C05501=1157.629,21.828,-48.363,-179.973,6.133,149.097
C05502=1157.624,22.077,-48.378,-179.970,6.134,149.096
C05503=1157.618,22.327,-48.393,-179.968,6.134,149.095
C05504=1157.613,22.576,-48.407,-179.966,6.135,149.095
C05505=1157.608,22.826,-48.421,-179.962,6.136,149.094
C05506=1157.603,23.076,-48.435,-179.960,6.137,149.094
C05507=1157.598,23.326,-48.450,-179.958,6.138,149.093
C05508=1157.593,23.575,-48.465,-179.955,6.138,149.093
C05509=1157.588,23.824,-48.479,-179.952,6.140,149.092
C05510=1157.583,24.074,-48.493,-179.950,6.140,149.092
C05511=1157.578,24.323,-48.507,-179.947,6.141,149.091
C05512=1157.573,24.573,-48.521,-179.945,6.142,149.090
C05513=1157.567,24.822,-48.537,-179.942,6.143,149.090
C05514=1157.562,25.072,-48.551,-179.940,6.144,149.089
C05515=1157.557,25.322,-48.566,-179.937,6.144,149.089
C05516=1157.552,25.571,-48.580,-179.935,6.145,149.088
C05517=1157.548,25.820,-48.595,-179.932,6.146,149.087
C05518=1157.543,26.070,-48.609,-179.930,6.147,149.087
C05519=1157.537,26.319,-48.624,-179.927,6.148,149.086
C05520=1157.532,26.569,-48.638,-179.924,6.149,149.086
C05521=1157.527,26.818,-48.653,-179.922,6.150,149.085
C05522=1157.522,27.068,-48.667,-179.919,6.151,149.085
C05523=1157.517,27.318,-48.681,-179.917,6.151,149.084
C05524=1157.511,27.587,-48.698,-179.914,6.153,149.084
C05525=1157.506,27.856,-48.713,-179.911,6.153,149.083
C05526=1157.501,28.124,-48.729,-179.908,6.155,149.082
C05527=1157.495,28.393,-48.745,-179.906,6.155,149.082
C05528=1157.490,28.643,-48.760,-179.903,6.156,149.081
C05529=1157.485,28.893,-48.774,-179.900,6.158,149.081
C05530=1157.481,29.142,-48.789,-179.898,6.158,149.080
C05531=1157.475,29.392,-48.804,-179.896,6.159,149.080
C05532=1157.470,29.640,-48.819,-179.892,6.160,149.079
C05533=1157.465,29.890,-48.833,-179.890,6.161,149.078
C05534=1157.460,30.140,-48.847,-179.888,6.161,149.078
C05535=1157.454,30.389,-48.863,-179.885,6.162,149.077
C05536=1157.449,30.639,-48.877,-179.882,6.164,149.077
C05537=1157.445,30.888,-48.892,-179.880,6.164,149.076
C05538=1157.439,31.138,-48.907,-179.877,6.165,149.076
C05539=1157.434,31.387,-48.922,-179.875,6.166,149.075
C05540=1157.429,31.637,-48.936,-179.872,6.167,149.074
C05541=1157.424,31.887,-48.950,-179.870,6.168,149.074
C05542=1157.419,32.136,-48.966,-179.867,6.169,149.073
C05543=1157.414,32.386,-48.980,-179.864,6.170,149.073
C05544=1157.409,32.635,-48.995,-179.862,6.170,149.072
C05545=1157.404,32.885,-49.010,-179.860,6.171,149.072
C05546=1157.399,33.134,-49.025,-179.856,6.172,149.071
C05547=1157.394,33.383,-49.040,-179.854,6.173,149.071
C05548=1157.389,33.633,-49.055,-179.852,6.174,149.070
C05549=1157.384,33.882,-49.070,-179.849,6.175,149.069
C05550=1157.378,34.132,-49.085,-179.846,6.176,149.069
C05551=1157.374,34.381,-49.100,-179.844,6.177,149.068
C05552=1157.369,34.631,-49.114,-179.841,6.178,149.068
C05553=1157.364,34.881,-49.130,-179.839,6.179,149.067
C05554=1157.359,35.131,-49.144,-179.836,6.179,149.066
C05555=1157.354,35.380,-49.160,-179.833,6.181,149.066
C05556=1157.349,35.629,-49.175,-179.831,6.182,149.066
C05557=1157.344,35.879,-49.189,-179.828,6.182,149.065
C05558=1157.339,36.128,-49.205,-179.826,6.184,149.064
C05559=1157.334,36.377,-49.220,-179.823,6.184,149.064
C05560=1157.328,36.627,-49.235,-179.821,6.185,149.063
C05561=1157.324,36.876,-49.250,-179.818,6.187,149.063
C05562=1157.318,37.126,-49.265,-179.815,6.187,149.062
C05563=1157.313,37.376,-49.279,-179.813,6.188,149.062
C05564=1157.308,37.625,-49.295,-179.810,6.190,149.061
C05565=1157.303,37.874,-49.310,-179.807,6.190,149.060
C05566=1157.298,38.124,-49.325,-179.805,6.191,149.060
C05567=1157.294,38.374,-49.340,-179.802,6.192,149.059
C05568=1157.288,38.623,-49.356,-179.800,6.193,149.059
C05569=1157.283,38.873,-49.370,-179.797,6.193,149.058
C05570=1157.278,39.122,-49.386,-179.794,6.195,149.058
C05571=1157.273,39.372,-49.401,-179.792,6.196,149.057
C05572=1157.268,39.621,-49.416,-179.790,6.196,149.057
C05573=1157.263,39.871,-49.431,-179.786,6.198,149.056
C05574=1157.257,40.120,-49.446,-179.784,6.199,149.055
C05575=1157.253,40.369,-49.461,-179.782,6.199,149.055
C05576=1157.248,40.619,-49.477,-179.779,6.201,149.054
C05577=1157.243,40.868,-49.492,-179.777,6.202,149.054
C05578=1157.238,41.118,-49.507,-179.774,6.202,149.053
C05579=1157.233,41.367,-49.522,-179.771,6.204,149.053
C05580=1157.228,41.617,-49.538,-179.769,6.204,149.052
C05581=1157.222,41.866,-49.553,-179.766,6.206,149.052
C05582=1157.218,42.116,-49.569,-179.763,6.206,149.051
C05583=1157.213,42.365,-49.584,-179.761,6.207,149.051
C05584=1157.208,42.615,-49.599,-179.758,6.208,149.050
C05585=1157.203,42.865,-49.614,-179.756,6.209,149.049
C05586=1157.197,43.114,-49.630,-179.753,6.210,149.049
C05587=1157.192,43.363,-49.645,-179.750,6.211,149.048
C05588=1157.188,43.613,-49.661,-179.748,6.212,149.048
C05589=1157.183,43.862,-49.676,-179.745,6.214,149.047
C05590=1157.178,44.112,-49.691,-179.743,6.214,149.047
C05591=1157.172,44.361,-49.707,-179.740,6.215,149.046
C05592=1157.168,44.610,-49.722,-179.737,6.217,149.046
C05593=1157.163,44.860,-49.738,-179.735,6.217,149.045
C05594=1157.157,45.110,-49.753,-179.733,6.218,149.045
C05595=1157.153,45.359,-49.768,-179.729,6.219,149.044
C05596=1157.147,45.608,-49.784,-179.727,6.220,149.043
C05597=1157.143,45.858,-49.800,-179.724,6.221,149.043
C05598=1157.138,46.107,-49.815,-179.722,6.222,149.042
C05599=1157.133,46.357,-49.830,-179.719,6.223,149.042
C05600=1157.127,46.606,-49.846,-179.716,6.224,149.041
C05601=1157.123,46.856,-49.861,-179.714,6.225,149.041
C05602=1157.118,47.105,-49.877,-179.711,6.226,149.040
C05603=1157.112,47.355,-49.892,-179.709,6.227,149.040
C05604=1157.107,47.604,-49.908,-179.706,6.228,149.039
C05605=1157.103,47.854,-49.923,-179.704,6.229,149.039
C05606=1157.098,48.103,-49.939,-179.701,6.230,149.038
C05607=1157.092,48.353,-49.955,-179.698,6.232,149.037
C05608=1157.088,48.602,-49.970,-179.695,6.232,149.037
C05609=1157.083,48.852,-49.986,-179.693,6.233,149.036
C05610=1157.077,49.101,-50.001,-179.690,6.234,149.036
C05611=1157.072,49.350,-50.017,-179.688,6.235,149.035
C05612=1157.068,49.600,-50.033,-179.685,6.237,149.035
C05613=1157.063,49.849,-50.048,-179.683,6.237,149.034
C05614=1157.057,50.099,-50.064,-179.680,6.239,149.034
C05615=1157.053,50.349,-50.080,-179.677,6.239,149.033
C05616=1157.047,50.598,-50.096,-179.675,6.240,149.033
C05617=1157.043,50.847,-50.110,-179.672,6.241,149.032
C05618=1157.038,51.096,-50.127,-179.670,6.242,149.031
C05619=1157.033,51.346,-50.143,-179.666,6.244,149.031
C05620=1157.027,51.596,-50.158,-179.664,6.244,149.030
C05621=1157.022,51.845,-50.174,-179.661,6.246,149.030
C05622=1157.018,52.094,-50.191,-179.659,6.247,149.029
C05623=1157.013,52.344,-50.206,-179.657,6.247,149.029
C05624=1157.008,52.594,-50.222,-179.653,6.249,149.028
C05625=1157.003,52.843,-50.237,-179.651,6.250,149.028
C05626=1156.998,53.092,-50.253,-179.648,6.251,149.027
C05627=1156.993,53.342,-50.269,-179.646,6.252,149.027
C05628=1156.987,53.610,-50.286,-179.643,6.253,149.026
C05629=1156.982,53.879,-50.303,-179.641,6.254,149.025
C05630=1156.976,54.147,-50.320,-179.637,6.255,149.025
C05631=1156.971,54.416,-50.337,-179.634,6.256,149.024
C05632=1156.966,54.666,-50.353,-179.632,6.257,149.024
C05633=1156.961,54.915,-50.370,-179.629,6.259,149.023
C05634=1156.957,55.165,-50.385,-179.627,6.259,149.023
C05635=1156.951,55.414,-50.401,-179.624,6.260,149.022
C05636=1156.946,55.663,-50.417,-179.621,6.262,149.021
C05637=1156.941,55.913,-50.433,-179.619,6.263,149.021
C05638=1156.936,56.162,-50.449,-179.616,6.264,149.021
C05639=1156.932,56.412,-50.465,-179.614,6.265,149.020
C05640=1156.926,56.661,-50.481,-179.611,6.266,149.019
C05641=1156.921,56.910,-50.497,-179.608,6.267,149.019
C05642=1156.916,57.160,-50.513,-179.605,6.268,149.018
C05643=1156.911,57.409,-50.529,-179.603,6.269,149.018
C05644=1156.906,57.659,-50.545,-179.600,6.271,149.017
C05645=1156.901,57.908,-50.561,-179.598,6.271,149.017
C05646=1156.897,58.158,-50.578,-179.595,6.273,149.016
C05647=1156.891,58.407,-50.593,-179.593,6.274,149.016
C05648=1156.887,58.657,-50.610,-179.589,6.275,149.015
C05649=1156.881,58.906,-50.625,-179.587,6.276,149.015
C05650=1156.876,59.155,-50.642,-179.584,6.277,149.014
C05651=1156.871,59.405,-50.658,-179.582,6.278,149.014
C05652=1156.866,59.654,-50.674,-179.580,6.279,149.013
C05653=1156.862,59.904,-50.690,-179.576,6.280,149.012
C05654=1156.856,60.153,-50.706,-179.574,6.281,149.012
C05655=1156.852,60.403,-50.722,-179.571,6.282,149.011
C05656=1156.847,60.652,-50.738,-179.569,6.283,149.011
C05657=1156.841,60.902,-50.755,-179.566,6.285,149.010
C05658=1156.836,61.151,-50.771,-179.564,6.285,149.010
C05659=1156.832,61.400,-50.788,-179.561,6.287,149.009
C05660=1156.826,61.650,-50.804,-179.558,6.287,149.009
C05661=1156.822,61.899,-50.820,-179.555,6.289,149.008
C05662=1156.816,62.148,-50.836,-179.553,6.290,149.008
C05663=1156.812,62.398,-50.852,-179.550,6.291,149.007
C05664=1156.807,62.647,-50.869,-179.548,6.292,149.007
C05665=1156.802,62.897,-50.885,-179.545,6.293,149.006
C05666=1156.796,63.146,-50.902,-179.542,6.294,149.006
C05667=1156.792,63.395,-50.918,-179.539,6.296,149.005
C05668=1156.787,63.646,-50.934,-179.537,6.296,149.005
C05669=1156.782,63.894,-50.951,-179.534,6.298,149.004
C05670=1156.777,64.144,-50.967,-179.532,6.299,149.003
C05671=1156.772,64.393,-50.983,-179.529,6.300,149.003
C05672=1156.767,64.643,-50.999,-179.526,6.301,149.002
C05673=1156.762,64.892,-51.016,-179.524,6.302,149.002
C05674=1156.757,65.142,-51.032,-179.521,6.304,149.001
C05675=1156.752,65.391,-51.049,-179.518,6.305,149.001
C05676=1156.747,65.640,-51.065,-179.516,6.306,149.000
C05677=1156.743,65.890,-51.082,-179.513,6.307,149.000
C05678=1156.737,66.139,-51.098,-179.510,6.308,148.999
C05679=1156.732,66.389,-51.115,-179.508,6.309,148.999
C05680=1156.727,66.638,-51.131,-179.505,6.311,148.998
C05681=1156.723,66.887,-51.148,-179.503,6.312,148.998
C05682=1156.717,67.137,-51.165,-179.500,6.313,148.997
C05683=1156.712,67.386,-51.181,-179.497,6.314,148.997
C05684=1156.708,67.636,-51.197,-179.494,6.315,148.996
C05685=1156.703,67.885,-51.214,-179.492,6.316,148.996
C05686=1156.697,68.134,-51.231,-179.489,6.318,148.995
C05687=1156.693,68.384,-51.248,-179.487,6.318,148.995
C05688=1156.688,68.633,-51.264,-179.484,6.320,148.994
C05689=1156.683,68.882,-51.281,-179.481,6.321,148.994
C05690=1156.678,69.133,-51.297,-179.478,6.322,148.993
C05691=1156.673,69.381,-51.313,-179.476,6.324,148.993
C05692=1156.668,69.631,-51.330,-179.473,6.324,148.992
C05693=1156.663,69.881,-51.347,-179.470,6.326,148.991
C05694=1156.658,70.129,-51.364,-179.468,6.327,148.991
C05695=1156.653,70.379,-51.380,-179.465,6.328,148.991
C05696=1156.648,70.629,-51.398,-179.463,6.329,148.990
C05697=1156.643,70.877,-51.414,-179.460,6.330,148.989
C05698=1156.639,71.127,-51.431,-179.457,6.332,148.989
C05699=1156.633,71.377,-51.448,-179.455,6.333,148.988
C05700=1156.628,71.625,-51.464,-179.452,6.334,148.988
C05701=1156.624,71.875,-51.481,-179.449,6.335,148.987
C05702=1156.619,72.125,-51.498,-179.447,6.336,148.987
C05703=1156.613,72.374,-51.514,-179.444,6.337,148.986
C05704=1156.608,72.623,-51.532,-179.441,6.339,148.986
C05705=1156.604,72.873,-51.548,-179.438,6.340,148.985
C05706=1156.599,73.122,-51.565,-179.436,6.341,148.985
C05707=1156.593,73.371,-51.582,-179.433,6.342,148.984
C05708=1156.589,73.621,-51.599,-179.431,6.343,148.984
C05709=1156.584,73.871,-51.616,-179.428,6.345,148.983
C05710=1156.579,74.119,-51.632,-179.426,6.346,148.983
C05711=1156.573,74.369,-51.649,-179.423,6.347,148.982
C05712=1156.569,74.619,-51.666,-179.420,6.349,148.982
C05713=1156.565,74.868,-51.683,-179.417,6.349,148.981
C05714=1156.559,75.117,-51.700,-179.415,6.351,148.981
C05715=1156.555,75.366,-51.717,-179.412,6.352,148.980
C05716=1156.549,75.616,-51.734,-179.409,6.353,148.980
C05717=1156.545,75.865,-51.751,-179.407,6.355,148.979
C05718=1156.539,76.115,-51.768,-179.404,6.355,148.979
C05719=1156.535,76.364,-51.784,-179.401,6.357,148.978
C05720=1156.530,76.613,-51.802,-179.399,6.358,148.978
C05721=1156.525,76.863,-51.819,-179.396,6.359,148.977
C05722=1156.520,77.113,-51.836,-179.393,6.361,148.977
C05723=1156.515,77.361,-51.853,-179.390,6.361,148.976
C05724=1156.510,77.611,-51.870,-179.388,6.363,148.976
C05725=1156.505,77.860,-51.887,-179.386,6.364,148.975
C05726=1156.500,78.110,-51.905,-179.382,6.365,148.975
C05727=1156.495,78.360,-51.922,-179.380,6.367,148.974
C05728=1156.490,78.608,-51.938,-179.378,6.368,148.974
C05729=1156.485,78.857,-51.956,-179.374,6.369,148.973
C05730=1156.481,79.107,-51.973,-179.372,6.370,148.973
C05731=1156.475,79.357,-51.990,-179.369,6.372,148.972
C05732=1156.470,79.625,-52.008,-179.366,6.373,148.971
C05733=1156.465,79.893,-52.027,-179.363,6.375,148.971
C05734=1156.460,80.162,-52.046,-179.361,6.375,148.970
C05735=1156.454,80.430,-52.064,-179.358,6.377,148.970
C05736=1156.449,80.679,-52.081,-179.355,6.378,148.969
C05737=1156.444,80.929,-52.099,-179.352,6.380,148.969
C05738=1156.440,81.178,-52.116,-179.350,6.381,148.968
C05739=1156.435,81.428,-52.133,-179.347,6.382,148.968
C05740=1156.430,81.677,-52.151,-179.345,6.383,148.967
C05741=1156.425,81.927,-52.167,-179.342,6.385,148.967
C05742=1156.420,82.175,-52.185,-179.339,6.386,148.966
C05743=1156.414,82.425,-52.202,-179.337,6.387,148.966
C05744=1156.410,82.674,-52.219,-179.334,6.389,148.965
C05745=1156.405,82.923,-52.237,-179.331,6.390,148.965
C05746=1156.400,83.173,-52.254,-179.328,6.391,148.964
C05747=1156.396,83.422,-52.272,-179.326,6.392,148.964
C05748=1156.390,83.672,-52.289,-179.322,6.394,148.963
C05749=1156.385,83.921,-52.307,-179.320,6.395,148.963
C05750=1156.381,84.171,-52.324,-179.318,6.396,148.962
C05751=1156.376,84.420,-52.342,-179.314,6.398,148.962
C05752=1156.370,84.669,-52.358,-179.312,6.399,148.961
C05753=1156.365,84.918,-52.376,-179.310,6.400,148.961
C05754=1156.361,85.168,-52.393,-179.306,6.402,148.960
C05755=1156.356,85.417,-52.411,-179.304,6.402,148.960
C05756=1156.351,85.666,-52.428,-179.301,6.404,148.959
C05757=1156.346,85.916,-52.446,-179.298,6.405,148.959
C05758=1156.341,86.165,-52.463,-179.296,6.406,148.958
C05759=1156.336,86.414,-52.481,-179.293,6.408,148.958
C05760=1156.332,86.663,-52.499,-179.291,6.410,148.958
C05761=1156.326,86.913,-52.516,-179.288,6.410,148.957
C05762=1156.321,87.162,-52.534,-179.285,6.412,148.956
C05763=1156.317,87.412,-52.551,-179.283,6.414,148.956
C05764=1156.312,87.661,-52.569,-179.280,6.414,148.955
C05765=1156.307,87.910,-52.587,-179.277,6.416,148.955
C05766=1156.302,88.160,-52.604,-179.274,6.417,148.955
C05767=1156.297,88.409,-52.622,-179.272,6.418,148.954
C05768=1156.293,88.658,-52.639,-179.269,6.420,148.954
C05769=1156.288,88.908,-52.657,-179.266,6.421,148.953
C05770=1156.283,89.157,-52.675,-179.264,6.422,148.952
C05771=1156.278,89.406,-52.693,-179.261,6.424,148.952
C05772=1156.273,89.656,-52.710,-179.258,6.425,148.952
C05773=1156.268,89.905,-52.728,-179.256,6.426,148.951
C05774=1156.263,90.154,-52.746,-179.253,6.427,148.951
C05775=1156.258,90.404,-52.764,-179.250,6.429,148.950
C05776=1156.253,90.653,-52.781,-179.248,6.430,148.950
C05777=1156.248,90.902,-52.799,-179.245,6.431,148.949
C05778=1156.243,91.151,-52.817,-179.242,6.433,148.949
C05779=1156.239,91.401,-52.834,-179.239,6.435,148.948
C05780=1156.233,91.650,-52.852,-179.237,6.436,148.948
C05781=1156.228,91.900,-52.870,-179.234,6.437,148.947
C05782=1156.224,92.149,-52.888,-179.231,6.439,148.947
C05783=1156.219,92.398,-52.906,-179.229,6.439,148.946
C05784=1156.214,92.647,-52.924,-179.226,6.441,148.946
C05785=1156.209,92.897,-52.941,-179.223,6.442,148.945
C05786=1156.204,93.147,-52.959,-179.220,6.444,148.945
C05787=1156.199,93.396,-52.977,-179.218,6.445,148.944
C05788=1156.194,93.645,-52.995,-179.215,6.446,148.944
C05789=1156.189,93.894,-53.013,-179.212,6.448,148.943
C05790=1156.185,94.143,-53.031,-179.210,6.449,148.943
C05791=1156.180,94.393,-53.049,-179.207,6.450,148.942
C05792=1156.175,94.642,-53.067,-179.204,6.452,148.942
C05793=1156.170,94.891,-53.085,-179.202,6.454,148.941
C05794=1156.165,95.141,-53.102,-179.199,6.455,148.941
C05795=1156.160,95.390,-53.120,-179.196,6.456,148.940
C05796=1156.155,95.640,-53.139,-179.193,6.458,148.940
C05797=1156.150,95.889,-53.157,-179.191,6.459,148.940
C05798=1156.146,96.138,-53.175,-179.189,6.460,148.939
C05799=1156.141,96.387,-53.193,-179.185,6.461,148.938
C05800=1156.136,96.637,-53.211,-179.183,6.463,148.938
C05801=1156.131,96.886,-53.229,-179.180,6.465,148.938
C05802=1156.126,97.135,-53.247,-179.178,6.466,148.937
C05803=1156.122,97.385,-53.265,-179.175,6.467,148.937
C05804=1156.117,97.634,-53.283,-179.172,6.469,148.936
C05805=1156.112,97.883,-53.301,-179.170,6.470,148.936
C05806=1156.106,98.133,-53.319,-179.167,6.471,148.935
C05807=1156.102,98.381,-53.338,-179.164,6.473,148.935
C05808=1156.097,98.630,-53.356,-179.161,6.474,148.934
C05809=1156.092,98.880,-53.375,-179.158,6.476,148.934
C05810=1156.087,99.129,-53.392,-179.156,6.477,148.933
C05811=1156.082,99.379,-53.410,-179.153,6.478,148.933
C05812=1156.078,99.628,-53.428,-179.150,6.480,148.932
C05813=1156.072,99.877,-53.447,-179.148,6.482,148.932
C05814=1156.068,100.127,-53.465,-179.145,6.483,148.932
C05815=1156.063,100.376,-53.483,-179.142,6.484,148.931
C05816=1156.058,100.625,-53.502,-179.139,6.486,148.931
C05817=1156.053,100.874,-53.520,-179.137,6.487,148.930
C05818=1156.048,101.123,-53.538,-179.135,6.488,148.930
C05819=1156.043,101.373,-53.557,-179.131,6.490,148.929
C05820=1156.038,101.623,-53.575,-179.129,6.491,148.929
C05821=1156.034,101.871,-53.594,-179.126,6.493,148.928
C05822=1156.029,102.120,-53.612,-179.123,6.495,148.928
C05823=1156.024,102.371,-53.631,-179.121,6.495,148.927
C05824=1156.019,102.620,-53.649,-179.118,6.497,148.927
C05825=1156.014,102.868,-53.667,-179.115,6.499,148.926
C05826=1156.009,103.117,-53.685,-179.112,6.500,148.926
C05827=1156.004,103.368,-53.704,-179.110,6.501,148.925
C05828=1155.999,103.617,-53.722,-179.107,6.502,148.925
C05829=1155.995,103.865,-53.741,-179.104,6.504,148.924
C05830=1155.990,104.114,-53.759,-179.102,6.506,148.924
C05831=1155.985,104.365,-53.778,-179.099,6.508,148.924
C05832=1155.980,104.613,-53.796,-179.096,6.508,148.923
C05833=1155.975,104.862,-53.814,-179.094,6.510,148.923
C05834=1155.970,105.113,-53.833,-179.091,6.511,148.922
C05835=1155.966,105.361,-53.852,-179.088,6.513,148.922
C05836=1155.960,105.629,-53.871,-179.085,6.514,148.921
C05837=1155.955,105.898,-53.891,-179.082,6.516,148.921
C05838=1155.951,106.166,-53.912,-179.079,6.518,148.920
C05839=1155.945,106.435,-53.932,-179.076,6.519,148.920
C05840=1155.940,106.684,-53.950,-179.074,6.521,148.919
C05841=1155.935,106.934,-53.970,-179.071,6.523,148.919
C05842=1155.930,107.183,-53.988,-179.068,6.523,148.918
C05843=1155.926,107.431,-54.006,-179.065,6.525,148.918
C05844=1155.920,107.682,-54.025,-179.063,6.527,148.917
C05845=1155.916,107.930,-54.044,-179.060,6.528,148.917
C05846=1155.911,108.179,-54.062,-179.057,6.530,148.917
C05847=1155.906,108.429,-54.081,-179.055,6.530,148.916
C05848=1155.901,108.678,-54.100,-179.052,6.532,148.916
C05849=1155.896,108.928,-54.118,-179.049,6.534,148.915
C05850=1155.892,109.177,-54.137,-179.047,6.536,148.915
C05851=1155.886,109.426,-54.156,-179.044,6.537,148.914
C05852=1155.882,109.676,-54.175,-179.041,6.539,148.914
C05853=1155.877,109.924,-54.193,-179.038,6.540,148.913
C05854=1155.872,110.174,-54.212,-179.036,6.541,148.913
C05855=1155.868,110.423,-54.231,-179.033,6.543,148.912
C05856=1155.862,110.672,-54.250,-179.030,6.545,148.912
C05857=1155.858,110.922,-54.269,-179.028,6.546,148.912
C05858=1155.853,111.170,-54.288,-179.024,6.548,148.911
C05859=1155.848,111.420,-54.306,-179.022,6.549,148.911
C05860=1155.843,111.669,-54.326,-179.020,6.550,148.910
C05861=1155.838,111.918,-54.344,-179.017,6.552,148.910
C05862=1155.833,112.168,-54.363,-179.014,6.554,148.909
C05863=1155.829,112.416,-54.382,-179.011,6.555,148.909
C05864=1155.824,112.667,-54.401,-179.008,6.557,148.908
C05865=1155.819,112.915,-54.420,-179.005,6.558,148.908
C05866=1155.814,113.164,-54.439,-179.003,6.559,148.908
C05867=1155.809,113.414,-54.458,-179.001,6.561,148.907
C05868=1155.804,113.663,-54.477,-178.998,6.563,148.907
C05869=1155.799,113.912,-54.496,-178.995,6.564,148.906
C05870=1155.795,114.161,-54.515,-178.992,6.566,148.906
C05871=1155.790,114.411,-54.534,-178.989,6.567,148.905
C05872=1155.785,114.660,-54.553,-178.987,6.569,148.905
C05873=1155.780,114.909,-54.572,-178.984,6.571,148.904
C05874=1155.775,115.158,-54.592,-178.982,6.572,148.904
C05875=1155.771,115.408,-54.610,-178.978,6.573,148.903
C05876=1155.765,115.657,-54.629,-178.976,6.575,148.903
C05877=1155.761,115.906,-54.649,-178.973,6.577,148.903
C05878=1155.756,116.155,-54.667,-178.970,6.578,148.902
C05879=1155.751,116.405,-54.687,-178.968,6.580,148.902
C05880=1155.747,116.653,-54.706,-178.965,6.582,148.901
C05881=1155.742,116.903,-54.725,-178.962,6.583,148.901
C05882=1155.736,117.152,-54.744,-178.960,6.584,148.900
C05883=1155.732,117.401,-54.763,-178.957,6.586,148.900
C05884=1155.727,117.650,-54.782,-178.954,6.587,148.900
C05885=1155.722,117.900,-54.802,-178.951,6.589,148.899
C05886=1155.718,118.148,-54.821,-178.949,6.591,148.899
C05887=1155.713,118.398,-54.840,-178.946,6.592,148.898
C05888=1155.708,118.648,-54.860,-178.943,6.594,148.898
C05889=1155.703,118.896,-54.879,-178.940,6.596,148.897
C05890=1155.699,119.146,-54.898,-178.937,6.597,148.897
C05891=1155.693,119.395,-54.918,-178.935,6.599,148.897
C05892=1155.689,119.644,-54.937,-178.932,6.600,148.896
C05893=1155.683,119.893,-54.957,-178.930,6.602,148.896
C05894=1155.679,120.142,-54.976,-178.927,6.603,148.895
C05895=1155.675,120.392,-54.995,-178.924,6.605,148.895
C05896=1155.669,120.641,-55.015,-178.921,6.606,148.894
C05897=1155.665,120.890,-55.034,-178.918,6.608,148.894
C05898=1155.660,121.139,-55.053,-178.916,6.610,148.893
C05899=1155.655,121.388,-55.073,-178.913,6.611,148.893
C05900=1155.650,121.638,-55.092,-178.910,6.613,148.893
C05901=1155.645,121.887,-55.112,-178.908,6.615,148.892
C05902=1155.640,122.136,-55.131,-178.905,6.617,148.892
C05903=1155.636,122.385,-55.150,-178.902,6.618,148.891
C05904=1155.631,122.634,-55.170,-178.899,6.619,148.891
C05905=1155.626,122.884,-55.189,-178.897,6.621,148.890
C05906=1155.621,123.133,-55.209,-178.894,6.622,148.890
C05907=1155.616,123.383,-55.228,-178.891,6.624,148.890
C05908=1155.612,123.631,-55.249,-178.889,6.626,148.889
C05909=1155.607,123.880,-55.267,-178.886,6.627,148.889
C05910=1155.602,124.130,-55.287,-178.883,6.629,148.888
C05911=1155.598,124.379,-55.307,-178.880,6.631,148.888
C05912=1155.592,124.628,-55.326,-178.877,6.632,148.887
C05913=1155.588,124.878,-55.346,-178.875,6.634,148.887
C05914=1155.583,125.127,-55.366,-178.872,6.636,148.887
C05915=1155.578,125.375,-55.385,-178.869,6.637,148.886
C05916=1155.573,125.625,-55.405,-178.866,6.639,148.886
C05917=1155.569,125.874,-55.424,-178.864,6.641,148.885
C05918=1155.564,126.122,-55.444,-178.861,6.642,148.885
C05919=1155.559,126.372,-55.464,-178.858,6.644,148.885
C05920=1155.554,126.622,-55.483,-178.856,6.646,148.884
C05921=1155.550,126.871,-55.503,-178.853,6.648,148.884
C05922=1155.545,127.119,-55.523,-178.850,6.648,148.883
C05923=1155.540,127.369,-55.543,-178.848,6.650,148.883
C05924=1155.535,127.619,-55.562,-178.845,6.652,148.882
C05925=1155.531,127.868,-55.583,-178.842,6.653,148.882
C05926=1155.525,128.116,-55.602,-178.839,6.655,148.882
C05927=1155.521,128.366,-55.622,-178.837,6.657,148.881
C05928=1155.516,128.615,-55.642,-178.834,6.658,148.881
C05929=1155.512,128.864,-55.662,-178.831,6.660,148.880
C05930=1155.506,129.113,-55.682,-178.829,6.662,148.880
C05931=1155.502,129.362,-55.701,-178.826,6.664,148.880
C05932=1155.497,129.612,-55.721,-178.823,6.665,148.879
C05933=1155.493,129.861,-55.741,-178.820,6.667,148.879
C05934=1155.487,130.110,-55.761,-178.817,6.668,148.878
C05935=1155.483,130.359,-55.781,-178.814,6.670,148.878
C05936=1155.478,130.608,-55.801,-178.812,6.672,148.877
C05937=1155.474,130.857,-55.821,-178.809,6.673,148.877
C05938=1155.468,131.107,-55.841,-178.806,6.675,148.877
C05939=1155.463,131.356,-55.861,-178.804,6.677,148.876
C05940=1155.458,131.624,-55.882,-178.801,6.679,148.876
C05941=1155.453,131.893,-55.903,-178.798,6.681,148.876
C05942=1155.448,132.162,-55.925,-178.794,6.682,148.875
C05943=1155.443,132.430,-55.947,-178.792,6.684,148.874
C05944=1155.437,132.679,-55.967,-178.789,6.686,148.874
C05945=1155.433,132.928,-55.988,-178.786,6.688,148.874
C05946=1155.428,133.178,-56.007,-178.784,6.689,148.873
C05947=1155.424,133.427,-56.028,-178.781,6.691,148.873
C05948=1155.419,133.675,-56.048,-178.778,6.693,148.873
C05949=1155.414,133.925,-56.067,-178.775,6.695,148.872
C05950=1155.410,134.174,-56.088,-178.773,6.696,148.872
C05951=1155.404,134.424,-56.108,-178.770,6.698,148.871
C05952=1155.400,134.672,-56.128,-178.767,6.700,148.871
C05953=1155.395,134.921,-56.149,-178.765,6.701,148.871
C05954=1155.391,135.171,-56.168,-178.762,6.703,148.870
C05955=1155.386,135.419,-56.188,-178.759,6.705,148.870
C05956=1155.380,135.668,-56.209,-178.756,6.707,148.869
C05957=1155.376,135.918,-56.229,-178.754,6.708,148.869
C05958=1155.371,136.167,-56.249,-178.751,6.710,148.869
C05959=1155.367,136.416,-56.270,-178.748,6.712,148.868
C05960=1155.362,136.665,-56.291,-178.746,6.713,148.868
C05961=1155.357,136.915,-56.310,-178.742,6.715,148.867
C05962=1155.352,137.164,-56.331,-178.740,6.717,148.867
C05963=1155.348,137.413,-56.351,-178.737,6.718,148.866
C05964=1155.343,137.662,-56.372,-178.734,6.720,148.866
C05965=1155.338,137.912,-56.392,-178.731,6.722,148.866
C05966=1155.333,138.160,-56.412,-178.728,6.724,148.865
C05967=1155.329,138.409,-56.432,-178.726,6.726,148.865
C05968=1155.323,138.658,-56.453,-178.723,6.728,148.865
C05969=1155.319,138.907,-56.473,-178.720,6.729,148.864
C05970=1155.314,139.156,-56.493,-178.717,6.731,148.864
C05971=1155.309,139.406,-56.514,-178.715,6.733,148.863
C05972=1155.305,139.655,-56.534,-178.712,6.735,148.863
C05973=1155.300,139.904,-56.555,-178.709,6.736,148.863
C05974=1155.295,140.153,-56.576,-178.707,6.738,148.862
C05975=1155.291,140.402,-56.596,-178.704,6.740,148.862
C05976=1155.286,140.651,-56.616,-178.701,6.741,148.861
C05977=1155.281,140.900,-56.637,-178.699,6.743,148.861
C05978=1155.276,141.150,-56.657,-178.696,6.745,148.861
C05979=1155.271,141.399,-56.678,-178.693,6.747,148.860
C05980=1155.267,141.648,-56.698,-178.690,6.748,148.860
C05981=1155.262,141.897,-56.719,-178.688,6.750,148.859
C05982=1155.257,142.146,-56.740,-178.684,6.753,148.859
C05983=1155.253,142.395,-56.760,-178.682,6.754,148.859
C05984=1155.247,142.644,-56.781,-178.679,6.756,148.858
C05985=1155.243,142.893,-56.801,-178.676,6.758,148.858
C05986=1155.238,143.142,-56.822,-178.674,6.759,148.858
C05987=1155.233,143.391,-56.843,-178.671,6.761,148.857
C05988=1155.229,143.640,-56.863,-178.668,6.763,148.857
C05989=1155.224,143.890,-56.884,-178.665,6.765,148.856
C05990=1155.219,144.139,-56.904,-178.663,6.766,148.856
C05991=1155.214,144.387,-56.926,-178.660,6.768,148.856
C05992=1155.211,144.637,-56.947,-178.657,6.770,148.855
C05993=1155.205,144.886,-56.968,-178.655,6.772,148.855
C05994=1155.201,145.135,-56.988,-178.652,6.774,148.855
C05995=1155.196,145.384,-57.009,-178.649,6.776,148.854
C05996=1155.191,145.633,-57.030,-178.646,6.778,148.854
C05997=1155.186,145.883,-57.051,-178.644,6.780,148.854
C05998=1155.182,146.131,-57.071,-178.641,6.781,148.853
C05999=1155.177,146.381,-57.092,-178.638,6.783,148.853
C06000=1155.172,146.629,-57.113,-178.636,6.785,148.852
C06001=1155.167,146.878,-57.134,-178.633,6.787,148.852
C06002=1155.162,147.128,-57.155,-178.630,6.788,148.852
C06003=1155.158,147.377,-57.176,-178.627,6.790,148.851
C06004=1155.153,147.627,-57.197,-178.624,6.792,148.851
C06005=1155.149,147.875,-57.218,-178.621,6.794,148.850
C06006=1155.144,148.124,-57.239,-178.619,6.796,148.850
C06007=1155.139,148.373,-57.260,-178.616,6.798,148.850
C06008=1155.134,148.622,-57.280,-178.613,6.799,148.849
C06009=1155.129,148.871,-57.302,-178.611,6.801,148.849
C06010=1155.125,149.120,-57.322,-178.608,6.803,148.849
C06011=1155.120,149.370,-57.343,-178.605,6.805,148.848
C06012=1155.115,149.618,-57.365,-178.602,6.807,148.848
C06013=1155.111,149.867,-57.385,-178.599,6.809,148.847
C06014=1155.106,150.117,-57.406,-178.597,6.811,148.847
C06015=1155.101,150.365,-57.428,-178.594,6.813,148.847
C06016=1155.096,150.614,-57.448,-178.592,6.814,148.847
C06017=1155.092,150.864,-57.470,-178.589,6.816,148.846
C06018=1155.087,151.113,-57.491,-178.586,6.818,148.846
C06019=1155.083,151.362,-57.512,-178.583,6.820,148.845
C06020=1155.077,151.611,-57.533,-178.580,6.822,148.845
C06021=1155.073,151.860,-57.554,-178.577,6.824,148.845
C06022=1155.068,152.110,-57.576,-178.575,6.826,148.844
C06023=1155.064,152.358,-57.597,-178.572,6.827,148.844
C06024=1155.059,152.607,-57.618,-178.569,6.829,148.843
C06025=1155.054,152.856,-57.640,-178.567,6.831,148.843
C06026=1155.049,153.105,-57.661,-178.563,6.833,148.843
C06027=1155.045,153.354,-57.682,-178.561,6.835,148.842
C06028=1155.040,153.603,-57.703,-178.558,6.837,148.842
C06029=1155.035,153.852,-57.725,-178.556,6.839,148.842
C06030=1155.030,154.101,-57.746,-178.553,6.841,148.841
C06031=1155.026,154.350,-57.767,-178.550,6.842,148.841
C06032=1155.021,154.600,-57.788,-178.547,6.845,148.841
C06033=1155.016,154.848,-57.810,-178.544,6.847,148.840
C06034=1155.011,155.098,-57.831,-178.542,6.848,148.840
C06035=1155.007,155.347,-57.853,-178.539,6.850,148.840
C06036=1155.002,155.596,-57.874,-178.536,6.852,148.839
C06037=1154.998,155.844,-57.895,-178.534,6.854,148.839
C06038=1154.993,156.094,-57.917,-178.531,6.856,148.839
C06039=1154.988,156.343,-57.938,-178.528,6.858,148.838
C06040=1154.983,156.592,-57.959,-178.525,6.860,148.838
C06041=1154.978,156.841,-57.980,-178.523,6.862,148.838
C06042=1154.974,157.090,-58.002,-178.520,6.863,148.837
C06043=1154.969,157.339,-58.024,-178.517,6.866,148.837
C06044=1154.964,157.608,-58.047,-178.514,6.868,148.836
C06045=1154.959,157.877,-58.070,-178.511,6.869,148.836
C06046=1154.954,158.146,-58.094,-178.508,6.872,148.836
C06047=1154.949,158.415,-58.117,-178.505,6.874,148.835
C06048=1154.945,158.664,-58.138,-178.503,6.875,148.835
C06049=1154.939,158.913,-58.159,-178.499,6.878,148.835
C06050=1154.935,159.162,-58.181,-178.497,6.880,148.834
C06051=1154.930,159.411,-58.203,-178.494,6.882,148.834
C06052=1154.926,159.660,-58.225,-178.492,6.883,148.834
C06053=1154.921,159.909,-58.246,-178.488,6.886,148.833
C06054=1154.916,160.158,-58.268,-178.486,6.888,148.833
C06055=1154.912,160.407,-58.290,-178.483,6.889,148.833
C06056=1154.907,160.656,-58.311,-178.480,6.891,148.832
C06057=1154.902,160.905,-58.333,-178.478,6.893,148.832
C06058=1154.898,161.154,-58.355,-178.474,6.896,148.831
C06059=1154.893,161.403,-58.376,-178.472,6.898,148.831
C06060=1154.888,161.653,-58.398,-178.469,6.899,148.831
C06061=1154.883,161.901,-58.420,-178.467,6.901,148.831
C06062=1154.879,162.150,-58.441,-178.464,6.903,148.830
C06063=1154.874,162.399,-58.463,-178.461,6.905,148.830
C06064=1154.869,162.648,-58.485,-178.458,6.907,148.829
C06065=1154.865,162.897,-58.507,-178.456,6.909,148.829
C06066=1154.860,163.146,-58.529,-178.453,6.911,148.829
C06067=1154.856,163.395,-58.551,-178.450,6.913,148.829
C06068=1154.850,163.644,-58.573,-178.447,6.915,148.828
C06069=1154.846,163.893,-58.595,-178.444,6.917,148.828
C06070=1154.841,164.142,-58.617,-178.442,6.919,148.827
C06071=1154.836,164.391,-58.639,-178.439,6.922,148.827
C06072=1154.832,164.640,-58.661,-178.436,6.923,148.827
C06073=1154.827,164.889,-58.682,-178.434,6.925,148.827
C06074=1154.823,165.138,-58.704,-178.431,6.927,148.826
C06075=1154.818,165.387,-58.726,-178.428,6.929,148.826
C06076=1154.814,165.636,-58.748,-178.425,6.931,148.825
C06077=1154.808,165.885,-58.770,-178.423,6.933,148.825
C06078=1154.804,166.134,-58.792,-178.420,6.935,148.825
C06079=1154.799,166.383,-58.814,-178.417,6.937,148.825
C06080=1154.795,166.632,-58.836,-178.414,6.939,148.824
C06081=1154.790,166.881,-58.858,-178.411,6.941,148.824
C06082=1154.786,167.130,-58.880,-178.409,6.943,148.824
C06083=1154.780,167.379,-58.902,-178.406,6.946,148.823
C06084=1154.776,167.628,-58.925,-178.403,6.947,148.823
C06085=1154.771,167.877,-58.947,-178.400,6.949,148.823
C06086=1154.767,168.126,-58.969,-178.398,6.951,148.822
C06087=1154.761,168.375,-58.991,-178.395,6.954,148.822
C06088=1154.757,168.624,-59.013,-178.392,6.955,148.822
C06089=1154.752,168.873,-59.035,-178.389,6.957,148.821
C06090=1154.748,169.122,-59.057,-178.387,6.959,148.821
C06091=1154.743,169.371,-59.080,-178.383,6.961,148.821
C06092=1154.738,169.620,-59.102,-178.381,6.964,148.820
C06093=1154.734,169.869,-59.124,-178.379,6.965,148.820
C06094=1154.730,170.117,-59.146,-178.375,6.968,148.820
C06095=1154.725,170.367,-59.169,-178.373,6.970,148.819
C06096=1154.720,170.616,-59.191,-178.370,6.971,148.819
C06097=1154.715,170.865,-59.213,-178.368,6.973,148.819
C06098=1154.710,171.113,-59.236,-178.364,6.976,148.819
C06099=1154.706,171.363,-59.258,-178.362,6.978,148.818
C06100=1154.702,171.612,-59.280,-178.359,6.979,148.818
C06101=1154.696,171.860,-59.303,-178.356,6.982,148.818
C06102=1154.692,172.110,-59.325,-178.354,6.984,148.817
C06103=1154.687,172.358,-59.347,-178.351,6.986,148.817
C06104=1154.682,172.607,-59.370,-178.348,6.988,148.817
C06105=1154.678,172.857,-59.392,-178.345,6.991,148.816
C06106=1154.674,173.105,-59.414,-178.343,6.992,148.816
C06107=1154.669,173.354,-59.437,-178.340,6.994,148.816
C06108=1154.665,173.603,-59.460,-178.337,6.997,148.815
C06109=1154.659,173.852,-59.482,-178.334,6.999,148.815
C06110=1154.655,174.101,-59.504,-178.332,7.000,148.815
C06111=1154.650,174.350,-59.527,-178.328,7.003,148.814
C06112=1154.645,174.599,-59.549,-178.326,7.005,148.814
C06113=1154.641,174.848,-59.572,-178.324,7.007,148.814
C06114=1154.636,175.097,-59.594,-178.320,7.009,148.814
C06115=1154.632,175.345,-59.617,-178.318,7.011,148.813
C06116=1154.627,175.595,-59.639,-178.315,7.013,148.813
C06117=1154.623,175.844,-59.662,-178.312,7.016,148.813
C06118=1154.617,176.093,-59.684,-178.309,7.017,148.812
C06119=1154.613,176.341,-59.707,-178.307,7.019,148.812
C06120=1154.608,176.590,-59.731,-178.303,7.022,148.812
C06121=1154.604,176.839,-59.752,-178.301,7.024,148.812
C06122=1154.599,177.088,-59.776,-178.299,7.026,148.811
C06123=1154.595,177.337,-59.798,-178.295,7.028,148.811
C06124=1154.590,177.586,-59.821,-178.293,7.030,148.811
C06125=1154.585,177.834,-59.843,-178.290,7.032,148.810
C06126=1154.580,178.084,-59.866,-178.287,7.035,148.810
C06127=1154.576,178.333,-59.889,-178.284,7.036,148.810
C06128=1154.571,178.581,-59.912,-178.282,7.038,148.809
C06129=1154.567,178.831,-59.934,-178.279,7.041,148.809
C06130=1154.562,179.080,-59.957,-178.276,7.043,148.809
C06131=1154.557,179.329,-59.981,-178.274,7.045,148.809
C06132=1154.553,179.578,-60.003,-178.271,7.047,148.808
C06133=1154.548,179.826,-60.026,-178.268,7.049,148.808
C06134=1154.544,180.075,-60.048,-178.265,7.051,148.808
C06135=1154.539,180.324,-60.072,-178.263,7.054,148.807
C06136=1154.534,180.574,-60.094,-178.260,7.056,148.807
C06137=1154.530,180.822,-60.117,-178.257,7.058,148.807
C06138=1154.525,181.071,-60.140,-178.254,7.060,148.807
C06139=1154.521,181.319,-60.163,-178.252,7.062,148.806
C06140=1154.516,181.568,-60.186,-178.248,7.064,148.806
C06141=1154.511,181.818,-60.209,-178.246,7.067,148.806
C06142=1154.507,182.066,-60.231,-178.243,7.068,148.805
C06143=1154.502,182.315,-60.255,-178.240,7.071,148.805
C06144=1154.497,182.564,-60.278,-178.238,7.073,148.805
C06145=1154.493,182.813,-60.301,-178.235,7.076,148.805
C06146=1154.489,183.062,-60.324,-178.232,7.077,148.804
C06147=1154.484,183.311,-60.348,-178.229,7.079,148.804
C06148=1154.479,183.581,-60.373,-178.227,7.082,148.804
C06149=1154.474,183.850,-60.397,-178.223,7.085,148.803
C06150=1154.469,184.120,-60.422,-178.221,7.086,148.803
C06151=1154.463,184.390,-60.447,-178.217,7.089,148.803
C06152=1154.459,184.638,-60.470,-178.215,7.091,148.803
C06153=1154.455,184.887,-60.493,-178.212,7.094,148.802
C06154=1154.450,185.137,-60.517,-178.209,7.095,148.802
C06155=1154.445,185.385,-60.540,-178.206,7.098,148.802
C06156=1154.441,185.634,-60.562,-178.204,7.100,148.801
C06157=1154.436,185.883,-60.586,-178.201,7.102,148.801
C06158=1154.431,186.132,-60.609,-178.198,7.105,148.801
C06159=1154.427,186.381,-60.632,-178.195,7.106,148.801
C06160=1154.422,186.630,-60.656,-178.192,7.109,148.800
C06161=1154.417,186.879,-60.679,-178.190,7.111,148.800
C06162=1154.414,187.127,-60.703,-178.187,7.113,148.800
C06163=1154.409,187.376,-60.726,-178.184,7.115,148.799
C06164=1154.404,187.625,-60.749,-178.182,7.117,148.799
C06165=1154.400,187.874,-60.773,-178.179,7.120,148.799
C06166=1154.394,188.122,-60.796,-178.176,7.122,148.799
C06167=1154.390,188.371,-60.819,-178.173,7.125,148.798
C06168=1154.385,188.620,-60.842,-178.170,7.126,148.798
C06169=1154.381,188.869,-60.865,-178.168,7.128,148.798
C06170=1154.376,189.117,-60.889,-178.165,7.131,148.798
C06171=1154.372,189.366,-60.913,-178.162,7.133,148.797
C06172=1154.367,189.616,-60.936,-178.159,7.136,148.797
C06173=1154.362,189.865,-60.959,-178.157,7.137,148.797
C06174=1154.358,190.114,-60.983,-178.154,7.140,148.797
C06175=1154.353,190.362,-61.007,-178.151,7.142,148.796
C06176=1154.349,190.611,-61.030,-178.149,7.144,148.796
C06177=1154.344,190.860,-61.053,-178.146,7.147,148.796
C06178=1154.339,191.109,-61.077,-178.143,7.149,148.795
C06179=1154.335,191.358,-61.101,-178.140,7.151,148.795
C06180=1154.330,191.607,-61.124,-178.138,7.153,148.795
C06181=1154.325,191.856,-61.148,-178.134,7.156,148.795
C06182=1154.321,192.104,-61.172,-178.132,7.158,148.795
C06183=1154.316,192.353,-61.195,-178.129,7.160,148.794
C06184=1154.312,192.602,-61.218,-178.127,7.163,148.794
C06185=1154.307,192.850,-61.242,-178.124,7.164,148.794
C06186=1154.302,193.099,-61.266,-178.121,7.167,148.793
C06187=1154.298,193.349,-61.289,-178.118,7.169,148.793
C06188=1154.293,193.597,-61.313,-178.115,7.172,148.793
C06189=1154.289,193.846,-61.337,-178.113,7.174,148.793
C06190=1154.284,194.094,-61.361,-178.110,7.176,148.792
C06191=1154.280,194.343,-61.384,-178.107,7.178,148.792
C06192=1154.275,194.592,-61.408,-178.104,7.181,148.792
C06193=1154.271,194.842,-61.432,-178.102,7.183,148.792
C06194=1154.266,195.091,-61.455,-178.099,7.186,148.792
C06195=1154.261,195.339,-61.480,-178.096,7.187,148.791
C06196=1154.257,195.588,-61.503,-178.093,7.190,148.791
C06197=1154.252,195.837,-61.527,-178.091,7.192,148.791
C06198=1154.247,196.086,-61.551,-178.088,7.195,148.791
C06199=1154.243,196.334,-61.575,-178.085,7.197,148.790
C06200=1154.239,196.583,-61.599,-178.082,7.198,148.790
C06201=1154.234,196.832,-61.622,-178.080,7.201,148.790
C06202=1154.230,197.080,-61.646,-178.077,7.203,148.789
C06203=1154.225,197.330,-61.671,-178.074,7.206,148.789
C06204=1154.220,197.579,-61.695,-178.071,7.208,148.789
C06205=1154.216,197.828,-61.718,-178.069,7.211,148.789
C06206=1154.211,198.076,-61.742,-178.066,7.212,148.789
C06207=1154.207,198.324,-61.766,-178.063,7.215,148.788
C06208=1154.201,198.574,-61.790,-178.061,7.217,148.788
C06209=1154.197,198.822,-61.814,-178.057,7.220,148.788
C06210=1154.193,199.071,-61.839,-178.055,7.222,148.788
C06211=1154.189,199.320,-61.862,-178.052,7.224,148.787
C06212=1154.184,199.569,-61.886,-178.050,7.226,148.787
C06213=1154.179,199.817,-61.911,-178.046,7.229,148.787
C06214=1154.174,200.066,-61.934,-178.044,7.231,148.787
C06215=1154.171,200.316,-61.959,-178.041,7.234,148.786
C06216=1154.166,200.564,-61.983,-178.039,7.236,148.786
C06217=1154.161,200.813,-62.007,-178.035,7.238,148.786
C06218=1154.156,201.062,-62.031,-178.033,7.241,148.786
C06219=1154.152,201.310,-62.055,-178.030,7.243,148.785
C06220=1154.147,201.560,-62.080,-178.027,7.246,148.785
C06221=1154.143,201.808,-62.104,-178.024,7.248,148.785
C06222=1154.139,202.056,-62.128,-178.022,7.251,148.785
C06223=1154.133,202.306,-62.152,-178.019,7.252,148.785
C06224=1154.129,202.554,-62.176,-178.016,7.255,148.784
C06225=1154.125,202.803,-62.200,-178.013,7.257,148.784
C06226=1154.120,203.052,-62.225,-178.011,7.260,148.784
C06227=1154.115,203.300,-62.249,-178.008,7.262,148.784
C06228=1154.112,203.550,-62.274,-178.005,7.265,148.784
C06229=1154.107,203.798,-62.298,-178.003,7.266,148.783
C06230=1154.102,204.047,-62.322,-178.000,7.269,148.783
C06231=1154.098,204.295,-62.346,-177.997,7.271,148.783
C06232=1154.093,204.544,-62.371,-177.994,7.274,148.783
C06233=1154.088,204.794,-62.395,-177.991,7.277,148.782
C06234=1154.083,205.042,-62.419,-177.989,7.279,148.782
C06235=1154.079,205.291,-62.444,-177.986,7.281,148.782
C06236=1154.074,205.540,-62.469,-177.983,7.283,148.782
C06237=1154.070,205.788,-62.493,-177.980,7.286,148.781
C06238=1154.065,206.037,-62.517,-177.978,7.288,148.781
C06239=1154.061,206.286,-62.542,-177.975,7.291,148.781
C06240=1154.057,206.535,-62.566,-177.972,7.293,148.781
C06241=1154.052,206.783,-62.591,-177.970,7.296,148.781
C06242=1154.048,207.032,-62.616,-177.966,7.298,148.780
C06243=1154.043,207.281,-62.640,-177.964,7.300,148.780
C06244=1154.039,207.529,-62.664,-177.961,7.303,148.780
C06245=1154.034,207.779,-62.689,-177.959,7.305,148.780
C06246=1154.029,208.027,-62.714,-177.955,7.308,148.780
C06247=1154.025,208.276,-62.738,-177.953,7.310,148.779
C06248=1154.020,208.525,-62.763,-177.950,7.312,148.779
C06249=1154.016,208.773,-62.787,-177.947,7.315,148.779
C06250=1154.011,209.022,-62.813,-177.944,7.317,148.779
C06251=1154.007,209.271,-62.837,-177.942,7.320,148.779
C06252=1154.002,209.541,-62.864,-177.938,7.323,148.778
C06253=1153.997,209.812,-62.891,-177.936,7.325,148.778
C06254=1153.992,210.082,-62.918,-177.933,7.327,148.778
C06255=1153.987,210.353,-62.945,-177.930,7.330,148.778
C06256=1153.982,210.602,-62.969,-177.927,7.333,148.777
C06257=1153.977,210.850,-62.994,-177.925,7.335,148.777
C06258=1153.974,211.099,-63.018,-177.922,7.338,148.777
C06259=1153.969,211.347,-63.044,-177.919,7.340,148.777
C06260=1153.964,211.597,-63.069,-177.916,7.342,148.777
C06261=1153.960,211.845,-63.093,-177.913,7.345,148.776
C06262=1153.955,212.093,-63.118,-177.911,7.347,148.776
C06263=1153.950,212.343,-63.143,-177.908,7.350,148.776
C06264=1153.946,212.591,-63.167,-177.905,7.353,148.776
C06265=1153.942,212.840,-63.193,-177.903,7.355,148.776
C06266=1153.937,213.089,-63.218,-177.899,7.357,148.775
C06267=1153.933,213.338,-63.242,-177.897,7.359,148.775
C06268=1153.928,213.586,-63.268,-177.894,7.362,148.775
C06269=1153.924,213.835,-63.293,-177.891,7.365,148.775
C06270=1153.919,214.083,-63.318,-177.889,7.367,148.775
C06271=1153.915,214.333,-63.343,-177.886,7.370,148.774
C06272=1153.910,214.581,-63.367,-177.883,7.373,148.774
C06273=1153.906,214.830,-63.393,-177.881,7.375,148.774
C06274=1153.901,215.079,-63.417,-177.878,7.377,148.774
C06275=1153.897,215.327,-63.443,-177.875,7.379,148.774
C06276=1153.892,215.576,-63.467,-177.872,7.382,148.774
C06277=1153.888,215.825,-63.493,-177.869,7.385,148.773
C06278=1153.882,216.074,-63.518,-177.867,7.387,148.773
C06279=1153.879,216.322,-63.543,-177.864,7.390,148.773
C06280=1153.874,216.571,-63.568,-177.861,7.392,148.773
C06281=1153.870,216.820,-63.593,-177.859,7.395,148.773
C06282=1153.865,217.068,-63.619,-177.856,7.397,148.772
C06283=1153.860,217.317,-63.644,-177.853,7.400,148.772
C06284=1153.856,217.565,-63.669,-177.850,7.402,148.772
C06285=1153.852,217.814,-63.694,-177.847,7.405,148.772
C06286=1153.847,218.062,-63.719,-177.845,7.407,148.772
C06287=1153.843,218.311,-63.745,-177.842,7.409,148.772
C06288=1153.838,218.561,-63.770,-177.839,7.412,148.771
C06289=1153.833,218.809,-63.795,-177.837,7.414,148.771
C06290=1153.829,219.058,-63.821,-177.834,7.417,148.771
C06291=1153.824,219.306,-63.846,-177.831,7.420,148.771
C06292=1153.820,219.555,-63.871,-177.829,7.422,148.771
C06293=1153.816,219.804,-63.897,-177.825,7.425,148.770
C06294=1153.811,220.052,-63.921,-177.823,7.428,148.770
C06295=1153.807,220.301,-63.947,-177.820,7.430,148.770
C06296=1153.802,220.549,-63.972,-177.817,7.432,148.770
C06297=1153.798,220.798,-63.998,-177.814,7.435,148.770
C06298=1153.793,221.047,-64.024,-177.812,7.437,148.770
C06299=1153.788,221.296,-64.049,-177.809,7.440,148.769
C06300=1153.784,221.544,-64.074,-177.806,7.443,148.769
C06301=1153.780,221.793,-64.100,-177.804,7.445,148.769
C06302=1153.775,222.041,-64.125,-177.801,7.448,148.769
C06303=1153.771,222.290,-64.151,-177.798,7.450,148.769
C06304=1153.766,222.539,-64.176,-177.795,7.453,148.769
C06305=1153.762,222.788,-64.202,-177.792,7.455,148.768
C06306=1153.757,223.036,-64.227,-177.790,7.458,148.768
C06307=1153.752,223.285,-64.253,-177.787,7.461,148.768
C06308=1153.748,223.533,-64.279,-177.784,7.463,148.768
C06309=1153.744,223.782,-64.304,-177.781,7.466,148.768
C06310=1153.740,224.031,-64.330,-177.779,7.469,148.768
C06311=1153.735,224.279,-64.355,-177.776,7.471,148.768
C06312=1153.731,224.528,-64.381,-177.773,7.473,148.767
C06313=1153.727,224.777,-64.407,-177.770,7.476,148.767
C06314=1153.722,225.025,-64.432,-177.768,7.478,148.767
C06315=1153.717,225.274,-64.459,-177.765,7.481,148.767
C06316=1153.712,225.523,-64.484,-177.762,7.484,148.767
C06317=1153.708,225.771,-64.510,-177.759,7.487,148.767
C06318=1153.703,226.020,-64.536,-177.757,7.489,148.766
C06319=1153.699,226.268,-64.561,-177.754,7.492,148.766
C06320=1153.695,226.517,-64.587,-177.751,7.494,148.766
C06321=1153.690,226.765,-64.612,-177.749,7.497,148.766
C06322=1153.685,227.014,-64.639,-177.746,7.499,148.766
C06323=1153.681,227.263,-64.664,-177.743,7.502,148.766
C06324=1153.677,227.512,-64.690,-177.740,7.505,148.766
C06325=1153.672,227.760,-64.716,-177.738,7.507,148.765
C06326=1153.668,228.009,-64.741,-177.735,7.510,148.765
C06327=1153.664,228.257,-64.768,-177.732,7.513,148.765
C06328=1153.659,228.506,-64.794,-177.729,7.516,148.765
C06329=1153.655,228.755,-64.820,-177.727,7.518,148.765
C06330=1153.650,229.003,-64.845,-177.724,7.520,148.765
C06331=1153.646,229.252,-64.871,-177.721,7.523,148.764
C06332=1153.641,229.500,-64.898,-177.718,7.526,148.764
C06333=1153.637,229.749,-64.924,-177.716,7.528,148.764
C06334=1153.632,229.998,-64.950,-177.713,7.531,148.764
C06335=1153.628,230.246,-64.975,-177.710,7.534,148.764
C06336=1153.623,230.495,-65.002,-177.707,7.537,148.764
C06337=1153.619,230.744,-65.028,-177.705,7.539,148.764
C06338=1153.615,230.992,-65.054,-177.702,7.541,148.763
C06339=1153.610,231.241,-65.080,-177.699,7.544,148.763
C06340=1153.605,231.489,-65.106,-177.696,7.547,148.763
C06341=1153.601,231.738,-65.132,-177.694,7.549,148.763
C06342=1153.596,231.987,-65.158,-177.691,7.552,148.763
C06343=1153.592,232.235,-65.185,-177.688,7.555,148.763
C06344=1153.588,232.484,-65.210,-177.685,7.558,148.763
C06345=1153.583,232.732,-65.237,-177.683,7.560,148.762
C06346=1153.579,232.981,-65.263,-177.680,7.563,148.762
C06347=1153.575,233.230,-65.289,-177.677,7.565,148.762
C06348=1153.569,233.478,-65.316,-177.674,7.568,148.762
C06349=1153.565,233.727,-65.341,-177.672,7.571,148.762
C06350=1153.561,233.975,-65.368,-177.669,7.573,148.762
C06351=1153.556,234.224,-65.394,-177.666,7.576,148.762
C06352=1153.552,234.472,-65.421,-177.663,7.579,148.761
C06353=1153.547,234.721,-65.447,-177.660,7.582,148.761
C06354=1153.543,234.969,-65.473,-177.658,7.584,148.761
C06355=1153.538,235.218,-65.500,-177.655,7.587,148.761
C06356=1153.534,235.490,-65.529,-177.652,7.590,148.761
C06357=1153.529,235.762,-65.557,-177.649,7.592,148.761
C06358=1153.524,236.033,-65.586,-177.646,7.596,148.761
C06359=1153.519,236.305,-65.615,-177.643,7.599,148.761
C06360=1153.515,236.554,-65.641,-177.640,7.601,148.760
C06361=1153.510,236.802,-65.668,-177.638,7.604,148.760
C06362=1153.506,237.051,-65.694,-177.635,7.607,148.760
C06363=1153.501,237.299,-65.721,-177.632,7.610,148.760
C06364=1153.497,237.548,-65.747,-177.629,7.613,148.760
C06365=1153.492,237.797,-65.774,-177.627,7.615,148.760
C06366=1153.489,238.045,-65.800,-177.624,7.617,148.760
C06367=1153.484,238.293,-65.827,-177.621,7.620,148.760
C06368=1153.479,238.543,-65.854,-177.618,7.623,148.760
C06369=1153.475,238.791,-65.880,-177.615,7.626,148.759
C06370=1153.470,239.039,-65.907,-177.613,7.628,148.759
C06371=1153.466,239.288,-65.933,-177.610,7.631,148.759
C06372=1153.461,239.536,-65.960,-177.607,7.634,148.759
C06373=1153.458,239.785,-65.986,-177.604,7.637,148.759
C06374=1153.453,240.033,-66.013,-177.602,7.640,148.759
C06375=1153.448,240.282,-66.040,-177.599,7.643,148.759
C06376=1153.444,240.530,-66.066,-177.597,7.645,148.759
C06377=1153.439,240.779,-66.093,-177.594,7.648,148.759
C06378=1153.435,241.027,-66.120,-177.591,7.651,148.758
C06379=1153.431,241.276,-66.147,-177.588,7.653,148.758
C06380=1153.426,241.524,-66.174,-177.585,7.656,148.758
C06381=1153.421,241.773,-66.200,-177.582,7.659,148.758
C06382=1153.417,242.021,-66.227,-177.580,7.661,148.758
C06383=1153.413,242.270,-66.254,-177.577,7.664,148.758
C06384=1153.409,242.519,-66.281,-177.575,7.667,148.758
C06385=1153.405,242.767,-66.308,-177.572,7.670,148.758
C06386=1153.400,243.016,-66.335,-177.569,7.673,148.758
C06387=1153.395,243.264,-66.362,-177.566,7.676,148.757
C06388=1153.391,243.512,-66.388,-177.564,7.678,148.757
C06389=1153.387,243.761,-66.415,-177.561,7.681,148.757
C06390=1153.382,244.009,-66.442,-177.558,7.684,148.757
C06391=1153.377,244.258,-66.469,-177.555,7.686,148.757
C06392=1153.374,244.506,-66.496,-177.552,7.689,148.757
C06393=1153.369,244.755,-66.523,-177.550,7.692,148.757
C06394=1153.365,245.004,-66.550,-177.547,7.694,148.757
C06395=1153.360,245.252,-66.577,-177.545,7.697,148.757
C06396=1153.355,245.501,-66.605,-177.541,7.700,148.756
C06397=1153.352,245.749,-66.631,-177.539,7.703,148.756
C06398=1153.347,245.998,-66.658,-177.536,7.706,148.756
C06399=1153.342,246.246,-66.685,-177.533,7.709,148.756
C06400=1153.338,246.495,-66.713,-177.530,7.712,148.756
C06401=1153.334,246.744,-66.740,-177.528,7.714,148.756
C06402=1153.329,246.992,-66.767,-177.525,7.717,148.756
C06403=1153.325,247.240,-66.794,-177.523,7.720,148.756
C06404=1153.321,247.488,-66.821,-177.520,7.723,148.756
C06405=1153.316,247.737,-66.848,-177.517,7.726,148.756
C06406=1153.312,247.986,-66.875,-177.514,7.728,148.756
C06407=1153.307,248.234,-66.902,-177.511,7.731,148.756
C06408=1153.303,248.482,-66.930,-177.509,7.734,148.756
C06409=1153.298,248.731,-66.957,-177.506,7.736,148.755
C06410=1153.294,248.979,-66.984,-177.503,7.739,148.755
C06411=1153.290,249.229,-67.012,-177.500,7.742,148.755
C06412=1153.285,249.476,-67.040,-177.498,7.745,148.755
C06413=1153.281,249.725,-67.066,-177.495,7.748,148.755
C06414=1153.277,249.973,-67.093,-177.492,7.751,148.755
C06415=1153.273,250.222,-67.121,-177.489,7.754,148.755
C06416=1153.268,250.470,-67.148,-177.487,7.757,148.755
C06417=1153.264,250.719,-67.175,-177.484,7.760,148.755
C06418=1153.259,250.967,-67.203,-177.482,7.762,148.755
C06419=1153.255,251.216,-67.231,-177.479,7.765,148.754
C06420=1153.250,251.464,-67.258,-177.476,7.768,148.754
C06421=1153.246,251.712,-67.285,-177.473,7.771,148.754
C06422=1153.241,251.961,-67.312,-177.470,7.774,148.754
C06423=1153.237,252.210,-67.340,-177.468,7.776,148.754
C06424=1153.233,252.458,-67.368,-177.465,7.779,148.754
C06425=1153.228,252.706,-67.395,-177.462,7.782,148.754
C06426=1153.224,252.955,-67.423,-177.459,7.785,148.754
C06427=1153.219,253.204,-67.451,-177.457,7.787,148.754
C06428=1153.215,253.451,-67.478,-177.454,7.790,148.754
C06429=1153.211,253.701,-67.506,-177.452,7.793,148.754
C06430=1153.207,253.948,-67.534,-177.449,7.796,148.754
C06431=1153.202,254.197,-67.561,-177.446,7.799,148.754
C06432=1153.198,254.446,-67.589,-177.443,7.802,148.754
C06433=1153.193,254.694,-67.616,-177.441,7.805,148.754
C06434=1153.189,254.942,-67.644,-177.438,7.808,148.753
C06435=1153.185,255.190,-67.672,-177.435,7.811,148.753
C06436=1153.180,255.439,-67.699,-177.432,7.814,148.753
C06437=1153.176,255.687,-67.727,-177.429,7.817,148.753
C06438=1153.172,255.936,-67.755,-177.427,7.820,148.753
C06439=1153.167,256.184,-67.782,-177.424,7.822,148.753
C06440=1153.163,256.432,-67.810,-177.422,7.825,148.753
C06441=1153.159,256.681,-67.838,-177.419,7.828,148.753
C06442=1153.154,256.930,-67.866,-177.416,7.831,148.753
C06443=1153.150,257.178,-67.894,-177.413,7.834,148.753
C06444=1153.145,257.427,-67.921,-177.411,7.837,148.753
C06445=1153.141,257.674,-67.949,-177.408,7.839,148.753
C06446=1153.137,257.923,-67.977,-177.405,7.842,148.753
C06447=1153.132,258.172,-68.005,-177.402,7.845,148.753
C06448=1153.128,258.420,-68.033,-177.399,7.848,148.753
C06449=1153.124,258.668,-68.061,-177.397,7.851,148.752
C06450=1153.119,258.917,-68.089,-177.394,7.854,148.752
C06451=1153.115,259.165,-68.117,-177.391,7.857,148.752
C06452=1153.110,259.414,-68.144,-177.389,7.860,148.752
C06453=1153.106,259.662,-68.172,-177.386,7.863,148.752
C06454=1153.101,259.910,-68.201,-177.383,7.866,148.752
C06455=1153.098,260.159,-68.229,-177.381,7.869,148.752
C06456=1153.093,260.407,-68.257,-177.378,7.871,148.752
C06457=1153.089,260.656,-68.285,-177.376,7.874,148.752
C06458=1153.084,260.904,-68.312,-177.373,7.877,148.752
C06459=1153.080,261.153,-68.341,-177.370,7.880,148.752
C06460=1153.076,261.426,-68.371,-177.367,7.884,148.752
C06461=1153.071,261.699,-68.403,-177.364,7.887,148.752
C06462=1153.066,261.972,-68.434,-177.361,7.890,148.752
C06463=1153.061,262.246,-68.465,-177.358,7.894,148.752
C06464=1153.056,262.494,-68.493,-177.355,7.896,148.752
C06465=1153.052,262.743,-68.521,-177.352,7.899,148.752
C06466=1153.048,262.990,-68.549,-177.349,7.902,148.752
C06467=1153.044,263.239,-68.578,-177.347,7.905,148.752
C06468=1153.039,263.487,-68.605,-177.344,7.908,148.752
C06469=1153.035,263.736,-68.634,-177.342,7.911,148.752
C06470=1153.030,263.984,-68.662,-177.339,7.914,148.752
C06471=1153.026,264.233,-68.691,-177.336,7.917,148.752
C06472=1153.022,264.481,-68.719,-177.333,7.920,148.752
C06473=1153.017,264.730,-68.747,-177.330,7.923,148.751
C06474=1153.013,264.978,-68.775,-177.328,7.925,148.751
C06475=1153.009,265.226,-68.804,-177.325,7.928,148.751
C06476=1153.005,265.474,-68.833,-177.323,7.931,148.751
C06477=1153.000,265.722,-68.861,-177.320,7.935,148.751
C06478=1152.996,265.971,-68.889,-177.318,7.937,148.751
C06479=1152.991,266.219,-68.917,-177.315,7.940,148.751
C06480=1152.987,266.468,-68.946,-177.312,7.943,148.751
C06481=1152.983,266.716,-68.975,-177.309,7.946,148.751
C06482=1152.979,266.964,-69.003,-177.307,7.949,148.751
C06483=1152.974,267.213,-69.032,-177.304,7.952,148.751
C06484=1152.970,267.461,-69.059,-177.301,7.955,148.751
C06485=1152.965,267.710,-69.088,-177.299,7.958,148.751
C06486=1152.961,267.958,-69.118,-177.296,7.961,148.751
C06487=1152.957,268.206,-69.145,-177.293,7.964,148.751
C06488=1152.952,268.455,-69.174,-177.290,7.967,148.751
C06489=1152.949,268.703,-69.203,-177.288,7.970,148.751
C06490=1152.944,268.951,-69.231,-177.285,7.973,148.751
C06491=1152.939,269.200,-69.260,-177.282,7.976,148.751
C06492=1152.936,269.448,-69.289,-177.280,7.979,148.751
C06493=1152.931,269.696,-69.317,-177.277,7.982,148.751
C06494=1152.926,269.945,-69.346,-177.274,7.985,148.751
C06495=1152.923,270.193,-69.375,-177.271,7.988,148.751
C06496=1152.918,270.441,-69.403,-177.269,7.991,148.751
C06497=1152.913,270.689,-69.433,-177.266,7.994,148.751
C06498=1152.910,270.938,-69.461,-177.264,7.997,148.751
C06499=1152.905,271.186,-69.489,-177.260,8.001,148.751
C06500=1152.900,271.434,-69.519,-177.257,8.004,148.751
C06501=1152.897,271.683,-69.547,-177.255,8.007,148.751
C06502=1152.892,271.930,-69.576,-177.252,8.010,148.751
C06503=1152.887,272.179,-69.605,-177.250,8.013,148.751
C06504=1152.883,272.427,-69.634,-177.247,8.016,148.751
C06505=1152.880,272.676,-69.662,-177.244,8.019,148.751
C06506=1152.875,272.924,-69.691,-177.241,8.022,148.751
C06507=1152.870,273.172,-69.720,-177.239,8.025,148.751
C06508=1152.866,273.421,-69.749,-177.236,8.028,148.751
C06509=1152.863,273.669,-69.778,-177.233,8.031,148.751
C06510=1152.858,273.917,-69.807,-177.231,8.034,148.751
C06511=1152.853,274.165,-69.836,-177.228,8.037,148.751
C06512=1152.849,274.414,-69.865,-177.226,8.040,148.751
C06513=1152.845,274.662,-69.894,-177.223,8.043,148.751
C06514=1152.841,274.910,-69.923,-177.220,8.046,148.751
C06515=1152.836,275.158,-69.952,-177.218,8.049,148.751
C06516=1152.832,275.407,-69.981,-177.215,8.052,148.751
C06517=1152.828,275.655,-70.010,-177.212,8.055,148.751
C06518=1152.823,275.904,-70.039,-177.209,8.058,148.751
C06519=1152.819,276.151,-70.068,-177.207,8.062,148.751
C06520=1152.814,276.400,-70.098,-177.204,8.065,148.751
C06521=1152.811,276.648,-70.127,-177.201,8.067,148.751
C06522=1152.806,276.897,-70.155,-177.199,8.070,148.751
C06523=1152.802,277.145,-70.185,-177.196,8.074,148.751
C06524=1152.798,277.393,-70.214,-177.194,8.077,148.751
C06525=1152.793,277.641,-70.243,-177.190,8.080,148.751
C06526=1152.789,277.889,-70.273,-177.188,8.083,148.751
C06527=1152.785,278.138,-70.302,-177.185,8.087,148.751
C06528=1152.780,278.386,-70.331,-177.182,8.090,148.751
C06529=1152.776,278.634,-70.360,-177.180,8.092,148.751
C06530=1152.772,278.883,-70.390,-177.177,8.096,148.751
C06531=1152.768,279.131,-70.419,-177.175,8.099,148.751
C06532=1152.763,279.378,-70.448,-177.172,8.102,148.751
C06533=1152.759,279.627,-70.478,-177.169,8.105,148.751
C06534=1152.755,279.875,-70.507,-177.167,8.108,148.751
C06535=1152.751,280.123,-70.537,-177.164,8.111,148.751
C06536=1152.746,280.372,-70.566,-177.161,8.114,148.751
C06537=1152.742,280.620,-70.595,-177.159,8.117,148.751
C06538=1152.738,280.869,-70.624,-177.156,8.120,148.751
C06539=1152.734,281.117,-70.654,-177.153,8.124,148.751
C06540=1152.729,281.365,-70.683,-177.150,8.127,148.751
C06541=1152.725,281.613,-70.712,-177.148,8.130,148.751
C06542=1152.720,281.861,-70.742,-177.145,8.133,148.751
C06543=1152.716,282.109,-70.771,-177.143,8.136,148.751
C06544=1152.712,282.357,-70.802,-177.140,8.139,148.751
C06545=1152.708,282.605,-70.831,-177.137,8.142,148.751
C06546=1152.704,282.853,-70.860,-177.134,8.145,148.751
C06547=1152.699,283.102,-70.890,-177.132,8.148,148.751
C06548=1152.695,283.350,-70.920,-177.129,8.151,148.751
C06549=1152.691,283.599,-70.949,-177.127,8.155,148.752
C06550=1152.686,283.847,-70.979,-177.124,8.157,148.751
C06551=1152.682,284.095,-71.008,-177.121,8.161,148.751
C06552=1152.678,284.343,-71.038,-177.118,8.164,148.752
C06553=1152.674,284.591,-71.069,-177.116,8.167,148.752
C06554=1152.669,284.840,-71.098,-177.113,8.170,148.752
C06555=1152.665,285.088,-71.127,-177.111,8.174,148.752
C06556=1152.661,285.336,-71.157,-177.108,8.177,148.752
C06557=1152.657,285.584,-71.187,-177.105,8.180,148.752
C06558=1152.652,285.832,-71.217,-177.103,8.183,148.752
C06559=1152.648,286.081,-71.247,-177.100,8.186,148.752
C06560=1152.644,286.329,-71.276,-177.097,8.190,148.752
C06561=1152.640,286.577,-71.306,-177.094,8.193,148.752
C06562=1152.636,286.825,-71.336,-177.092,8.196,148.752
C06563=1152.631,287.073,-71.366,-177.089,8.199,148.752
C06564=1152.626,287.348,-71.399,-177.086,8.202,148.752
C06565=1152.621,287.624,-71.432,-177.083,8.206,148.752
C06566=1152.617,287.899,-71.465,-177.080,8.210,148.752
C06567=1152.612,288.174,-71.498,-177.077,8.213,148.752
C06568=1152.608,288.422,-71.529,-177.075,8.216,148.752
C06569=1152.603,288.671,-71.558,-177.072,8.219,148.752
C06570=1152.600,288.918,-71.588,-177.069,8.223,148.752
C06571=1152.595,289.167,-71.618,-177.067,8.226,148.753
C06572=1152.591,289.415,-71.648,-177.064,8.229,148.752
C06573=1152.587,289.663,-71.678,-177.062,8.232,148.753
C06574=1152.583,289.911,-71.709,-177.059,8.235,148.753
C06575=1152.578,290.160,-71.739,-177.056,8.238,148.753
C06576=1152.575,290.407,-71.769,-177.054,8.241,148.753
C06577=1152.570,290.656,-71.799,-177.051,8.244,148.753
C06578=1152.566,290.904,-71.829,-177.048,8.248,148.753
C06579=1152.562,291.152,-71.858,-177.045,8.251,148.753
C06580=1152.557,291.400,-71.889,-177.043,8.255,148.753
C06581=1152.553,291.648,-71.919,-177.040,8.258,148.753
C06582=1152.549,291.897,-71.950,-177.037,8.261,148.753
C06583=1152.545,292.145,-71.979,-177.035,8.264,148.753
C06584=1152.540,292.393,-72.010,-177.032,8.267,148.753
C06585=1152.536,292.641,-72.040,-177.029,8.271,148.753
C06586=1152.532,292.889,-72.070,-177.027,8.274,148.753
C06587=1152.527,293.137,-72.100,-177.024,8.277,148.753
C06588=1152.524,293.385,-72.131,-177.022,8.280,148.753
C06589=1152.519,293.634,-72.161,-177.019,8.283,148.754
C06590=1152.515,293.881,-72.191,-177.017,8.286,148.754
C06591=1152.511,294.129,-72.222,-177.014,8.290,148.754
C06592=1152.507,294.377,-72.252,-177.011,8.293,148.754
C06593=1152.502,294.626,-72.282,-177.009,8.297,148.754
C06594=1152.499,294.874,-72.313,-177.006,8.300,148.754
C06595=1152.494,295.122,-72.343,-177.003,8.303,148.754
C06596=1152.489,295.370,-72.374,-177.001,8.306,148.754
C06597=1152.485,295.618,-72.404,-176.998,8.309,148.754
C06598=1152.481,295.867,-72.435,-176.995,8.313,148.754
C06599=1152.477,296.114,-72.465,-176.993,8.316,148.754
C06600=1152.473,296.362,-72.496,-176.990,8.319,148.754
C06601=1152.469,296.610,-72.526,-176.988,8.322,148.754
C06602=1152.465,296.859,-72.557,-176.985,8.325,148.754
C06603=1152.460,297.107,-72.587,-176.982,8.329,148.755
C06604=1152.456,297.355,-72.617,-176.979,8.332,148.755
C06605=1152.451,297.603,-72.648,-176.977,8.336,148.755
C06606=1152.447,297.852,-72.679,-176.974,8.339,148.755
C06607=1152.443,298.099,-72.709,-176.972,8.342,148.755
C06608=1152.439,298.347,-72.740,-176.969,8.345,148.755
C06609=1152.436,298.595,-72.770,-176.966,8.349,148.755
C06610=1152.431,298.843,-72.801,-176.963,8.352,148.755
C06611=1152.426,299.091,-72.832,-176.961,8.355,148.755
C06612=1152.422,299.340,-72.863,-176.959,8.358,148.755
C06613=1152.418,299.588,-72.893,-176.956,8.361,148.755
C06614=1152.414,299.836,-72.924,-176.953,8.365,148.756
C06615=1152.409,300.084,-72.955,-176.950,8.368,148.756
C06616=1152.406,300.332,-72.985,-176.948,8.372,148.756
C06617=1152.401,300.580,-73.016,-176.945,8.375,148.756
C06618=1152.397,300.828,-73.047,-176.943,8.378,148.756
C06619=1152.393,301.077,-73.078,-176.940,8.382,148.756
C06620=1152.389,301.324,-73.109,-176.937,8.385,148.756
C06621=1152.385,301.572,-73.140,-176.935,8.388,148.756
C06622=1152.381,301.820,-73.171,-176.932,8.391,148.756
C06623=1152.376,302.068,-73.202,-176.930,8.394,148.756
C06624=1152.372,302.317,-73.233,-176.927,8.398,148.756
C06625=1152.368,302.564,-73.263,-176.924,8.401,148.757
C06626=1152.364,302.812,-73.294,-176.922,8.405,148.757
C06627=1152.360,303.060,-73.325,-176.919,8.408,148.757
C06628=1152.355,303.308,-73.356,-176.917,8.411,148.757
C06629=1152.350,303.556,-73.387,-176.913,8.415,148.757
C06630=1152.346,303.805,-73.418,-176.911,8.418,148.757
C06631=1152.342,304.052,-73.450,-176.909,8.421,148.757
C06632=1152.339,304.301,-73.480,-176.906,8.424,148.757
C06633=1152.334,304.549,-73.511,-176.903,8.428,148.758
C06634=1152.330,304.796,-73.542,-176.901,8.432,148.758
C06635=1152.326,305.045,-73.574,-176.898,8.435,148.758
C06636=1152.321,305.293,-73.604,-176.896,8.438,148.758
C06637=1152.318,305.541,-73.636,-176.893,8.441,148.758
C06638=1152.313,305.789,-73.667,-176.890,8.445,148.758
C06639=1152.309,306.037,-73.698,-176.888,8.448,148.758
C06640=1152.305,306.285,-73.730,-176.885,8.451,148.758
C06641=1152.301,306.533,-73.761,-176.883,8.454,148.758
C06642=1152.296,306.781,-73.792,-176.880,8.458,148.759
C06643=1152.292,307.029,-73.823,-176.877,8.461,148.759
C06644=1152.288,307.277,-73.854,-176.875,8.465,148.759
C06645=1152.283,307.525,-73.885,-176.872,8.468,148.759
C06646=1152.279,307.773,-73.917,-176.869,8.472,148.759
C06647=1152.275,308.021,-73.948,-176.867,8.475,148.759
C06648=1152.271,308.269,-73.979,-176.864,8.478,148.759
C06649=1152.267,308.517,-74.011,-176.862,8.481,148.759
C06650=1152.263,308.765,-74.042,-176.859,8.484,148.760
C06651=1152.258,309.013,-74.073,-176.856,8.489,148.760
C06652=1152.255,309.261,-74.105,-176.854,8.492,148.760
C06653=1152.250,309.509,-74.136,-176.851,8.495,148.760
C06654=1152.246,309.757,-74.168,-176.849,8.498,148.760
C06655=1152.242,310.005,-74.199,-176.846,8.502,148.760
C06656=1152.238,310.253,-74.230,-176.843,8.505,148.760
C06657=1152.234,310.501,-74.262,-176.841,8.508,148.760
C06658=1152.230,310.749,-74.293,-176.838,8.512,148.761
C06659=1152.225,310.997,-74.325,-176.835,8.515,148.761
C06660=1152.221,311.244,-74.357,-176.833,8.519,148.761
C06661=1152.217,311.493,-74.388,-176.831,8.522,148.761
C06662=1152.213,311.740,-74.420,-176.828,8.526,148.761
C06663=1152.209,311.988,-74.451,-176.825,8.529,148.761
C06664=1152.205,312.237,-74.483,-176.823,8.532,148.761
C06665=1152.201,312.484,-74.514,-176.821,8.536,148.762
C06666=1152.196,312.733,-74.546,-176.817,8.539,148.762
C06667=1152.192,312.980,-74.578,-176.815,8.543,148.762
C06668=1152.188,313.258,-74.614,-176.812,8.547,148.762
C06669=1152.183,313.536,-74.648,-176.809,8.551,148.762
C06670=1152.179,313.813,-74.684,-176.806,8.554,148.762
C06671=1152.174,314.090,-74.719,-176.803,8.558,148.762
C06672=1152.169,314.338,-74.752,-176.801,8.561,148.763
C06673=1152.166,314.586,-74.784,-176.798,8.565,148.763
C06674=1152.161,314.834,-74.815,-176.795,8.568,148.763
C06675=1152.158,315.082,-74.847,-176.793,8.571,148.763
C06676=1152.152,315.330,-74.878,-176.790,8.576,148.763
C06677=1152.149,315.578,-74.910,-176.788,8.579,148.763
C06678=1152.145,315.826,-74.942,-176.785,8.582,148.763
C06679=1152.140,316.074,-74.974,-176.783,8.585,148.764
C06680=1152.136,316.322,-75.006,-176.780,8.589,148.764
C06681=1152.132,316.570,-75.038,-176.778,8.592,148.764
C06682=1152.129,316.818,-75.070,-176.775,8.596,148.764
C06683=1152.124,317.066,-75.102,-176.772,8.599,148.764
C06684=1152.120,317.314,-75.133,-176.770,8.603,148.764
C06685=1152.116,317.562,-75.165,-176.767,8.606,148.765
C06686=1152.111,317.809,-75.197,-176.765,8.609,148.765
C06687=1152.107,318.057,-75.229,-176.762,8.613,148.765
C06688=1152.104,318.305,-75.261,-176.759,8.616,148.765
C06689=1152.100,318.553,-75.294,-176.757,8.620,148.765
C06690=1152.095,318.800,-75.326,-176.754,8.624,148.765
C06691=1152.091,319.049,-75.358,-176.752,8.627,148.766
C06692=1152.087,319.297,-75.390,-176.749,8.630,148.766
C06693=1152.083,319.545,-75.422,-176.747,8.634,148.766
C06694=1152.078,319.792,-75.454,-176.744,8.637,148.766
C06695=1152.075,320.041,-75.486,-176.741,8.641,148.766
C06696=1152.071,320.288,-75.519,-176.739,8.645,148.767
C06697=1152.067,320.536,-75.551,-176.736,8.648,148.767
C06698=1152.062,320.784,-75.583,-176.734,8.651,148.767
C06699=1152.058,321.032,-75.615,-176.731,8.655,148.767
C06700=1152.054,321.280,-75.648,-176.729,8.659,148.767
C06701=1152.050,321.528,-75.680,-176.726,8.662,148.767
C06702=1152.046,321.776,-75.712,-176.723,8.666,148.768
C06703=1152.042,322.023,-75.744,-176.721,8.669,148.768
C06704=1152.037,322.271,-75.777,-176.718,8.672,148.768
C06705=1152.034,322.519,-75.809,-176.716,8.676,148.768
C06706=1152.029,322.768,-75.841,-176.713,8.680,148.768
C06707=1152.026,323.015,-75.874,-176.711,8.683,148.769
C06708=1152.021,323.263,-75.906,-176.708,8.687,148.769
C06709=1152.017,323.511,-75.937,-176.705,8.690,148.769
C06710=1152.013,323.758,-75.971,-176.703,8.693,148.769
C06711=1152.009,324.006,-76.002,-176.700,8.697,148.769
C06712=1152.005,324.254,-76.036,-176.698,8.700,148.769
C06713=1152.001,324.502,-76.067,-176.695,8.704,148.770
C06714=1151.997,324.750,-76.101,-176.692,8.708,148.770
C06715=1151.992,324.998,-76.133,-176.690,8.711,148.770
C06716=1151.989,325.245,-76.165,-176.688,8.714,148.770
C06717=1151.984,325.493,-76.198,-176.685,8.718,148.770
C06718=1151.980,325.741,-76.231,-176.683,8.722,148.771
C06719=1151.977,325.989,-76.263,-176.680,8.725,148.771
C06720=1151.972,326.237,-76.296,-176.677,8.729,148.771
C06721=1151.968,326.485,-76.328,-176.675,8.732,148.771
C06722=1151.965,326.733,-76.361,-176.672,8.735,148.771
C06723=1151.960,326.981,-76.393,-176.669,8.739,148.771
C06724=1151.956,327.229,-76.426,-176.667,8.743,148.772
C06725=1151.952,327.476,-76.458,-176.664,8.747,148.772
C06726=1151.948,327.724,-76.491,-176.662,8.750,148.772
C06727=1151.943,327.971,-76.524,-176.660,8.753,148.772
C06728=1151.940,328.220,-76.556,-176.657,8.757,148.773
C06729=1151.936,328.467,-76.589,-176.654,8.761,148.773
C06730=1151.931,328.715,-76.622,-176.652,8.764,148.773
C06731=1151.927,328.963,-76.655,-176.649,8.768,148.773
C06732=1151.924,329.211,-76.687,-176.647,8.771,148.773
C06733=1151.919,329.458,-76.721,-176.644,8.775,148.774
C06734=1151.915,329.706,-76.754,-176.642,8.779,148.774
C06735=1151.911,329.955,-76.786,-176.639,8.782,148.774
C06736=1151.907,330.202,-76.819,-176.636,8.786,148.774
C06737=1151.903,330.450,-76.852,-176.634,8.789,148.774
C06738=1151.899,330.697,-76.885,-176.632,8.793,148.775
C06739=1151.895,330.946,-76.917,-176.629,8.797,148.775
C06740=1151.891,331.194,-76.951,-176.627,8.800,148.775
C06741=1151.886,331.441,-76.984,-176.624,8.804,148.775
C06742=1151.882,331.689,-77.017,-176.621,8.807,148.776
C06743=1151.878,331.937,-77.050,-176.619,8.811,148.776
C06744=1151.875,332.184,-77.083,-176.616,8.815,148.776
C06745=1151.871,332.432,-77.116,-176.614,8.818,148.776
C06746=1151.866,332.680,-77.148,-176.611,8.822,148.776
C06747=1151.862,332.928,-77.181,-176.609,8.825,148.777
C06748=1151.858,333.176,-77.215,-176.606,8.829,148.777
C06749=1151.854,333.423,-77.248,-176.603,8.833,148.777
C06750=1151.850,333.671,-77.281,-176.601,8.836,148.777
C06751=1151.845,333.919,-77.314,-176.598,8.840,148.777
C06752=1151.841,334.167,-77.347,-176.596,8.843,148.778
C06753=1151.837,334.414,-77.380,-176.593,8.847,148.778
C06754=1151.833,334.662,-77.414,-176.591,8.851,148.778
C06755=1151.829,334.910,-77.447,-176.588,8.854,148.778
C06756=1151.825,335.158,-77.480,-176.585,8.858,148.779
C06757=1151.821,335.406,-77.513,-176.583,8.861,148.779
C06758=1151.817,335.654,-77.547,-176.580,8.866,148.779
C06759=1151.813,335.901,-77.580,-176.578,8.869,148.779
C06760=1151.809,336.148,-77.614,-176.576,8.872,148.780
C06761=1151.805,336.396,-77.647,-176.573,8.876,148.780
C06762=1151.801,336.644,-77.680,-176.571,8.880,148.780
C06763=1151.797,336.892,-77.713,-176.568,8.884,148.780
C06764=1151.793,337.139,-77.746,-176.565,8.887,148.780
C06765=1151.789,337.388,-77.780,-176.563,8.891,148.781
C06766=1151.785,337.635,-77.814,-176.560,8.894,148.781
C06767=1151.781,337.883,-77.847,-176.558,8.898,148.781
C06768=1151.777,338.130,-77.880,-176.555,8.902,148.781
C06769=1151.773,338.378,-77.913,-176.553,8.905,148.782
C06770=1151.769,338.625,-77.947,-176.550,8.910,148.782
C06771=1151.765,338.874,-77.980,-176.548,8.913,148.782
C06772=1151.760,339.154,-78.019,-176.545,8.917,148.782
C06773=1151.756,339.434,-78.056,-176.542,8.921,148.783
C06774=1151.752,339.713,-78.094,-176.539,8.925,148.783
C06775=1151.747,339.994,-78.132,-176.536,8.929,148.783
C06776=1151.743,340.242,-78.166,-176.533,8.933,148.783
C06777=1151.739,340.490,-78.199,-176.532,8.937,148.784
C06778=1151.735,340.737,-78.233,-176.529,8.941,148.784
C06779=1151.730,340.985,-78.266,-176.526,8.944,148.784
C06780=1151.726,341.233,-78.300,-176.523,8.948,148.785
C06781=1151.722,341.480,-78.334,-176.521,8.952,148.785
C06782=1151.718,341.728,-78.367,-176.518,8.956,148.785
C06783=1151.714,341.975,-78.401,-176.516,8.959,148.785
C06784=1151.710,342.224,-78.435,-176.513,8.963,148.786
C06785=1151.706,342.471,-78.469,-176.511,8.967,148.786
C06786=1151.702,342.719,-78.502,-176.509,8.970,148.786
C06787=1151.698,342.966,-78.536,-176.506,8.974,148.786
C06788=1151.694,343.214,-78.570,-176.504,8.977,148.787
C06789=1151.690,343.462,-78.604,-176.501,8.981,148.787
C06790=1151.686,343.709,-78.637,-176.499,8.985,148.787
C06791=1151.682,343.957,-78.671,-176.496,8.989,148.787
C06792=1151.678,344.205,-78.705,-176.494,8.992,148.788
C06793=1151.674,344.452,-78.739,-176.491,8.996,148.788
C06794=1151.670,344.700,-78.773,-176.488,9.000,148.788
C06795=1151.665,344.947,-78.806,-176.486,9.004,148.789
C06796=1151.662,345.195,-78.841,-176.484,9.007,148.789
C06797=1151.657,345.443,-78.874,-176.481,9.011,148.789
C06798=1151.654,345.690,-78.908,-176.478,9.015,148.789
C06799=1151.650,345.939,-78.943,-176.475,9.019,148.790
C06800=1151.646,346.186,-78.977,-176.474,9.022,148.790
C06801=1151.642,346.433,-79.010,-176.471,9.026,148.790
C06802=1151.638,346.681,-79.045,-176.468,9.030,148.790
C06803=1151.634,346.929,-79.079,-176.465,9.034,148.791
C06804=1151.629,347.177,-79.113,-176.463,9.037,148.791
C06805=1151.626,347.424,-79.147,-176.461,9.042,148.791
C06806=1151.621,347.672,-79.181,-176.458,9.045,148.792
C06807=1151.617,347.919,-79.215,-176.455,9.049,148.792
C06808=1151.614,348.167,-79.249,-176.453,9.052,148.792
C06809=1151.609,348.415,-79.283,-176.451,9.057,148.792
C06810=1151.606,348.663,-79.317,-176.448,9.060,148.793
C06811=1151.601,348.910,-79.352,-176.445,9.064,148.793
C06812=1151.598,349.157,-79.386,-176.443,9.068,148.793
C06813=1151.594,349.405,-79.421,-176.441,9.072,148.794
C06814=1151.590,349.652,-79.454,-176.438,9.075,148.794
C06815=1151.586,349.900,-79.489,-176.435,9.079,148.794
C06816=1151.582,350.148,-79.523,-176.433,9.083,148.794
C06817=1151.577,350.395,-79.558,-176.431,9.087,148.795
C06818=1151.574,350.643,-79.591,-176.428,9.091,148.795
C06819=1151.569,350.891,-79.626,-176.425,9.094,148.795
C06820=1151.565,351.139,-79.660,-176.423,9.098,148.796
C06821=1151.561,351.386,-79.694,-176.421,9.102,148.796
C06822=1151.558,351.634,-79.729,-176.418,9.106,148.796
C06823=1151.554,351.881,-79.764,-176.416,9.109,148.796
C06824=1151.549,352.128,-79.798,-176.413,9.113,148.797
C06825=1151.545,352.376,-79.833,-176.411,9.117,148.797
C06826=1151.542,352.623,-79.867,-176.408,9.121,148.797
C06827=1151.538,352.871,-79.902,-176.406,9.124,148.798
C06828=1151.534,353.119,-79.936,-176.403,9.129,148.798
C06829=1151.530,353.367,-79.970,-176.401,9.132,148.798
C06830=1151.525,353.614,-80.005,-176.398,9.136,148.799
C06831=1151.522,353.862,-80.039,-176.395,9.140,148.799
C06832=1151.517,354.109,-80.074,-176.393,9.144,148.799
C06833=1151.514,354.357,-80.109,-176.390,9.148,148.799
C06834=1151.510,354.604,-80.143,-176.388,9.151,148.800
C06835=1151.506,354.852,-80.178,-176.385,9.155,148.800
C06836=1151.501,355.100,-80.212,-176.383,9.159,148.800
C06837=1151.498,355.347,-80.247,-176.380,9.163,148.801
C06838=1151.495,355.595,-80.282,-176.378,9.167,148.801
C06839=1151.490,355.842,-80.317,-176.375,9.171,148.801
C06840=1151.486,356.090,-80.351,-176.373,9.175,148.802
C06841=1151.482,356.337,-80.386,-176.371,9.178,148.802
C06842=1151.479,356.585,-80.421,-176.368,9.182,148.802
C06843=1151.474,356.832,-80.455,-176.365,9.186,148.802
C06844=1151.470,357.080,-80.491,-176.363,9.190,148.803
C06845=1151.466,357.327,-80.525,-176.360,9.194,148.803
C06846=1151.462,357.575,-80.560,-176.358,9.197,148.803
C06847=1151.459,357.823,-80.595,-176.355,9.202,148.804
C06848=1151.454,358.070,-80.630,-176.353,9.205,148.804
C06849=1151.450,358.318,-80.664,-176.350,9.210,148.805
C06850=1151.447,358.565,-80.699,-176.348,9.214,148.805
C06851=1151.443,358.813,-80.734,-176.345,9.217,148.805
C06852=1151.439,359.060,-80.769,-176.343,9.221,148.805
C06853=1151.435,359.308,-80.804,-176.340,9.225,148.806
C06854=1151.431,359.555,-80.839,-176.338,9.229,148.806
C06855=1151.427,359.803,-80.874,-176.335,9.233,148.806
C06856=1151.423,360.050,-80.909,-176.333,9.236,148.807
C06857=1151.419,360.298,-80.944,-176.330,9.240,148.807
C06858=1151.416,360.545,-80.979,-176.327,9.245,148.807
C06859=1151.411,360.793,-81.014,-176.325,9.248,148.808
C06860=1151.408,361.040,-81.049,-176.323,9.253,148.808
C06861=1151.404,361.288,-81.085,-176.320,9.257,148.808
C06862=1151.399,361.535,-81.119,-176.317,9.260,148.809
C06863=1151.396,361.783,-81.155,-176.315,9.264,148.809
C06864=1151.392,362.030,-81.190,-176.312,9.268,148.809
C06865=1151.387,362.278,-81.225,-176.310,9.272,148.810
C06866=1151.384,362.525,-81.260,-176.307,9.276,148.810
C06867=1151.380,362.773,-81.296,-176.304,9.280,148.810
C06868=1151.376,363.020,-81.330,-176.302,9.285,148.811
C06869=1151.372,363.268,-81.366,-176.299,9.288,148.811
C06870=1151.368,363.515,-81.401,-176.297,9.292,148.811
C06871=1151.364,363.763,-81.436,-176.294,9.296,148.812
C06872=1151.360,364.010,-81.471,-176.292,9.300,148.812
C06873=1151.356,364.258,-81.507,-176.289,9.304,148.812
C06874=1151.353,364.505,-81.543,-176.286,9.308,148.813
C06875=1151.349,364.753,-81.578,-176.284,9.312,148.813
C06876=1151.344,365.035,-81.619,-176.281,9.317,148.813
C06877=1151.340,365.319,-81.658,-176.279,9.321,148.814
C06878=1151.336,365.602,-81.699,-176.275,9.326,148.814
C06879=1151.331,365.885,-81.739,-176.273,9.330,148.815
C06880=1151.327,366.132,-81.775,-176.270,9.334,148.815
C06881=1151.323,366.380,-81.810,-176.267,9.339,148.815
C06882=1151.320,366.627,-81.846,-176.265,9.342,148.816
C06883=1151.315,366.875,-81.882,-176.262,9.346,148.816
C06884=1151.311,367.122,-81.917,-176.259,9.351,148.816
C06885=1151.307,367.370,-81.953,-176.257,9.355,148.817
C06886=1151.304,367.617,-81.988,-176.255,9.359,148.817
C06887=1151.300,367.865,-82.024,-176.252,9.363,148.817
C06888=1151.296,368.112,-82.059,-176.250,9.367,148.818
C06889=1151.291,368.359,-82.095,-176.247,9.371,148.818
C06890=1151.288,368.607,-82.131,-176.245,9.375,148.819
C06891=1151.284,368.854,-82.166,-176.242,9.379,148.819
C06892=1151.280,369.102,-82.202,-176.239,9.383,148.819
C06893=1151.277,369.349,-82.237,-176.238,9.387,148.820
C06894=1151.272,369.597,-82.273,-176.235,9.391,148.820
C06895=1151.269,369.844,-82.309,-176.233,9.396,148.821
C06896=1151.265,370.091,-82.345,-176.230,9.400,148.821
C06897=1151.261,370.338,-82.380,-176.228,9.403,148.821
C06898=1151.256,370.586,-82.417,-176.225,9.408,148.822
C06899=1151.253,370.833,-82.452,-176.223,9.412,148.822
C06900=1151.249,371.081,-82.488,-176.221,9.416,148.823
C06901=1151.245,371.328,-82.525,-176.218,9.420,148.823
C06902=1151.241,371.576,-82.560,-176.216,9.424,148.824
C06903=1151.238,371.823,-82.596,-176.214,9.428,148.824
C06904=1151.233,372.071,-82.632,-176.211,9.432,148.824
C06905=1151.229,372.318,-82.667,-176.209,9.436,148.825
C06906=1151.226,372.565,-82.703,-176.207,9.440,148.825
C06907=1151.221,372.812,-82.739,-176.204,9.444,148.826
C06908=1151.218,373.060,-82.775,-176.202,9.449,148.826
C06909=1151.214,373.307,-82.811,-176.200,9.453,148.827
C06910=1151.210,373.555,-82.847,-176.198,9.457,148.827
C06911=1151.206,373.802,-82.883,-176.196,9.461,148.828
C06912=1151.203,374.049,-82.919,-176.194,9.465,148.828
C06913=1151.198,374.297,-82.955,-176.192,9.469,148.829
C06914=1151.195,374.544,-82.992,-176.190,9.473,148.829
C06915=1151.191,374.792,-83.028,-176.188,9.477,148.830
C06916=1151.187,375.039,-83.063,-176.185,9.481,148.830
C06917=1151.183,375.286,-83.100,-176.184,9.485,148.831
C06918=1151.179,375.534,-83.136,-176.181,9.490,148.831
C06919=1151.176,375.781,-83.172,-176.180,9.494,148.832
C06920=1151.172,376.028,-83.208,-176.177,9.498,148.832
C06921=1151.168,376.275,-83.244,-176.176,9.502,148.833
C06922=1151.164,376.523,-83.280,-176.174,9.505,148.833
C06923=1151.160,376.770,-83.317,-176.172,9.510,148.834
C06924=1151.156,377.018,-83.353,-176.170,9.514,148.834
C06925=1151.153,377.265,-83.389,-176.168,9.518,148.835
C06926=1151.148,377.512,-83.425,-176.166,9.522,148.836
C06927=1151.145,377.759,-83.462,-176.165,9.526,148.836
C06928=1151.141,378.007,-83.498,-176.163,9.530,148.837
C06929=1151.136,378.254,-83.535,-176.162,9.534,148.837
C06930=1151.133,378.501,-83.571,-176.160,9.538,148.838
C06931=1151.129,378.749,-83.607,-176.158,9.542,148.839
C06932=1151.125,378.996,-83.643,-176.157,9.546,148.839
C06933=1151.121,379.243,-83.680,-176.155,9.550,148.840
C06934=1151.118,379.491,-83.716,-176.154,9.554,148.841
C06935=1151.113,379.738,-83.752,-176.152,9.558,148.841
C06936=1151.109,379.985,-83.789,-176.151,9.562,148.842
C06937=1151.106,380.232,-83.825,-176.150,9.566,148.843
C06938=1151.102,380.480,-83.862,-176.148,9.570,148.843
C06939=1151.098,380.727,-83.898,-176.147,9.574,148.844
C06940=1151.094,380.975,-83.934,-176.146,9.577,148.845
C06941=1151.090,381.222,-83.971,-176.145,9.581,148.845
C06942=1151.087,381.469,-84.008,-176.143,9.585,148.846
C06943=1151.083,381.716,-84.044,-176.142,9.589,148.847
C06944=1151.079,381.964,-84.080,-176.141,9.592,148.847
C06945=1151.075,382.211,-84.117,-176.140,9.596,148.848
C06946=1151.071,382.458,-84.154,-176.140,9.600,148.849
C06947=1151.068,382.705,-84.190,-176.138,9.604,148.849
C06948=1151.064,382.952,-84.227,-176.138,9.607,148.850
C06949=1151.059,383.200,-84.263,-176.137,9.611,148.851
C06950=1151.056,383.448,-84.300,-176.136,9.615,148.852
C06951=1151.052,383.695,-84.336,-176.135,9.618,148.852
C06952=1151.048,383.942,-84.373,-176.134,9.622,148.853
C06953=1151.045,384.189,-84.410,-176.134,9.625,148.854
C06954=1151.041,384.436,-84.446,-176.133,9.629,148.855
C06955=1151.036,384.684,-84.483,-176.133,9.632,148.855
C06956=1151.032,384.931,-84.519,-176.132,9.635,148.856
C06957=1151.030,385.179,-84.556,-176.132,9.639,148.857
C06958=1151.025,385.426,-84.593,-176.132,9.642,148.858
C06959=1151.021,385.673,-84.630,-176.131,9.646,148.859
C06960=1151.018,385.920,-84.666,-176.131,9.649,148.859
C06961=1151.014,386.167,-84.703,-176.132,9.652,148.860
C06962=1151.010,386.414,-84.740,-176.131,9.655,148.861
C06963=1151.006,386.662,-84.777,-176.131,9.659,148.862
C06964=1151.003,386.909,-84.813,-176.131,9.662,148.863
C06965=1150.999,387.157,-84.849,-176.131,9.665,148.863
C06966=1150.994,387.404,-84.886,-176.131,9.668,148.864
C06967=1150.990,387.651,-84.923,-176.131,9.671,148.865
C06968=1150.987,387.898,-84.959,-176.131,9.674,148.866
C06969=1150.983,388.145,-84.996,-176.131,9.677,148.867
C06970=1150.979,388.393,-85.033,-176.131,9.681,148.868
C06971=1150.976,388.640,-85.070,-176.131,9.683,148.868
C06972=1150.972,388.887,-85.107,-176.132,9.686,148.869
C06973=1150.968,389.135,-85.143,-176.132,9.689,148.870
C06974=1150.964,389.382,-85.180,-176.133,9.691,148.871
C06975=1150.960,389.629,-85.217,-176.133,9.694,148.872
C06976=1150.957,389.877,-85.254,-176.134,9.697,148.873
C06977=1150.953,390.124,-85.291,-176.134,9.700,148.873
C06978=1150.949,390.371,-85.328,-176.134,9.703,148.874
C06979=1150.945,390.618,-85.364,-176.135,9.705,148.875
C06980=1150.940,390.905,-85.407,-176.135,9.708,148.876
C06981=1150.936,391.191,-85.450,-176.136,9.712,148.877
C06982=1150.932,391.478,-85.492,-176.137,9.714,148.878
C06983=1150.928,391.764,-85.535,-176.137,9.717,148.879
C06984=1150.924,392.011,-85.572,-176.138,9.720,148.880
C06985=1150.920,392.258,-85.608,-176.138,9.723,148.881
C06986=1150.916,392.505,-85.645,-176.140,9.725,148.882
C06987=1150.912,392.752,-85.682,-176.140,9.728,148.882
C06988=1150.909,393.000,-85.719,-176.141,9.731,148.883
C06989=1150.904,393.247,-85.756,-176.141,9.733,148.884
C06990=1150.901,393.494,-85.792,-176.142,9.735,148.885
C06991=1150.897,393.741,-85.829,-176.143,9.737,148.886
C06992=1150.893,393.989,-85.866,-176.143,9.740,148.887
C06993=1150.889,394.237,-85.903,-176.145,9.742,148.888
C06994=1150.885,394.484,-85.940,-176.146,9.744,148.888
C06995=1150.882,394.731,-85.976,-176.146,9.747,148.889
C06996=1150.878,394.978,-86.013,-176.147,9.749,148.890
C06997=1150.874,395.225,-86.050,-176.148,9.751,148.891
C06998=1150.870,395.472,-86.087,-176.149,9.754,148.892
C06999=1150.866,395.720,-86.124,-176.150,9.756,148.892
C07000=1150.863,395.967,-86.161,-176.151,9.758,148.893
C07001=1150.859,396.214,-86.197,-176.151,9.761,148.894
C07002=1150.855,396.461,-86.234,-176.152,9.763,148.895
C07003=1150.851,396.709,-86.271,-176.154,9.765,148.896
C07004=1150.847,396.956,-86.308,-176.155,9.767,148.897
C07005=1150.843,397.204,-86.345,-176.155,9.769,148.897
C07006=1150.840,397.450,-86.382,-176.156,9.771,148.898
C07007=1150.836,397.697,-86.419,-176.157,9.774,148.899
C07008=1150.832,397.944,-86.456,-176.158,9.776,148.900
C07009=1150.828,398.192,-86.493,-176.159,9.778,148.901
C07010=1150.824,398.439,-86.530,-176.160,9.780,148.902
C07011=1150.821,398.686,-86.566,-176.161,9.782,148.902
C07012=1150.817,398.933,-86.603,-176.162,9.784,148.903
C07013=1150.813,399.181,-86.640,-176.163,9.786,148.904
C07014=1150.809,399.429,-86.677,-176.164,9.788,148.905
C07015=1150.805,399.676,-86.714,-176.165,9.790,148.906
C07016=1150.801,399.923,-86.751,-176.166,9.792,148.906
C07017=1150.798,400.170,-86.787,-176.167,9.794,148.907
C07018=1150.793,400.417,-86.824,-176.168,9.796,148.908
C07019=1150.790,400.665,-86.861,-176.169,9.798,148.909
C07020=1150.786,400.912,-86.898,-176.170,9.800,148.909
C07021=1150.782,401.159,-86.935,-176.171,9.802,148.910
C07022=1150.778,401.406,-86.971,-176.172,9.804,148.911
C07023=1150.774,401.653,-87.008,-176.173,9.806,148.912
C07024=1150.771,401.901,-87.046,-176.174,9.808,148.913
C07025=1150.767,402.148,-87.083,-176.175,9.810,148.913
C07026=1150.763,402.395,-87.120,-176.176,9.812,148.914
C07027=1150.759,402.642,-87.157,-176.177,9.814,148.915
C07028=1150.755,402.889,-87.193,-176.178,9.816,148.916
C07029=1150.752,403.137,-87.230,-176.179,9.818,148.917
C07030=1150.748,403.384,-87.267,-176.180,9.819,148.917
C07031=1150.744,403.631,-87.304,-176.181,9.821,148.918
C07032=1150.740,403.879,-87.341,-176.182,9.823,148.919
C07033=1150.736,404.126,-87.378,-176.183,9.825,148.920
C07034=1150.733,404.373,-87.414,-176.184,9.827,148.920
C07035=1150.729,404.620,-87.451,-176.185,9.829,148.921
C07036=1150.725,404.868,-87.488,-176.186,9.830,148.922
C07037=1150.721,405.115,-87.525,-176.187,9.832,148.922
C07038=1150.716,405.362,-87.562,-176.188,9.834,148.923
C07039=1150.714,405.609,-87.599,-176.189,9.836,148.924
C07040=1150.710,405.856,-87.636,-176.190,9.838,148.925
C07041=1150.706,406.103,-87.673,-176.191,9.840,148.925
C07042=1150.702,406.351,-87.710,-176.192,9.842,148.926
C07043=1150.698,406.598,-87.746,-176.192,9.844,148.927
C07044=1150.694,406.846,-87.784,-176.193,9.846,148.928
C07045=1150.691,407.093,-87.820,-176.194,9.847,148.928
C07046=1150.687,407.340,-87.857,-176.195,9.849,148.929
C07047=1150.683,407.587,-87.894,-176.196,9.851,148.930
C07048=1150.678,407.834,-87.930,-176.197,9.853,148.930
C07049=1150.675,408.082,-87.968,-176.198,9.855,148.931
C07050=1150.671,408.329,-88.005,-176.198,9.857,148.932
C07051=1150.668,408.576,-88.041,-176.199,9.859,148.933
C07052=1150.663,408.823,-88.078,-176.200,9.861,148.933
C07053=1150.660,409.070,-88.115,-176.201,9.862,148.934
C07054=1150.656,409.318,-88.152,-176.202,9.864,148.935
C07055=1150.652,409.565,-88.189,-176.203,9.866,148.936
C07056=1150.648,409.812,-88.226,-176.203,9.868,148.936
C07057=1150.645,410.059,-88.262,-176.204,9.870,148.937
C07058=1150.641,410.306,-88.299,-176.205,9.872,148.938
C07059=1150.637,410.554,-88.337,-176.206,9.873,148.938
C07060=1150.633,410.801,-88.373,-176.206,9.875,148.939
C07061=1150.629,411.048,-88.410,-176.207,9.877,148.940
C07062=1150.625,411.296,-88.447,-176.208,9.879,148.940
C07063=1150.621,411.542,-88.483,-176.209,9.881,148.941
C07064=1150.618,411.790,-88.521,-176.210,9.882,148.942
C07065=1150.614,412.038,-88.557,-176.211,9.885,148.943
C07066=1150.610,412.284,-88.595,-176.211,9.886,148.943
C07067=1150.606,412.531,-88.632,-176.212,9.888,148.944
C07068=1150.602,412.779,-88.669,-176.213,9.890,148.944
C07069=1150.598,413.026,-88.706,-176.213,9.892,148.945
C07070=1150.595,413.273,-88.742,-176.214,9.893,148.946
C07071=1150.591,413.520,-88.779,-176.215,9.895,148.947
C07072=1150.587,413.768,-88.816,-176.215,9.898,148.947
C07073=1150.583,414.015,-88.853,-176.216,9.900,148.948
C07074=1150.579,414.263,-88.890,-176.217,9.901,148.949
C07075=1150.575,414.510,-88.927,-176.217,9.903,148.949
C07076=1150.572,414.756,-88.964,-176.218,9.905,148.950
C07077=1150.569,415.004,-89.001,-176.219,9.907,148.950
C07078=1150.566,415.252,-89.038,-176.219,9.908,148.951
C07079=1150.564,415.498,-89.074,-176.219,9.911,148.952
C07080=1150.564,415.718,-89.107,-176.220,9.913,148.952
C07081=1150.563,415.938,-89.139,-176.221,9.915,148.953
C07082=1150.563,416.159,-89.172,-176.221,9.916,148.954
C07083=1150.564,416.377,-89.204,-176.222,9.918,148.954
C07084=1150.565,416.597,-89.236,-176.222,9.919,148.955
C07085=1150.568,416.817,-89.268,-176.223,9.921,148.955
C07086=1150.570,417.037,-89.300,-176.223,9.922,148.956
C07087=1150.573,417.256,-89.333,-176.224,9.923,148.956
C07088=1150.153,417.257,-89.381,-176.226,9.935,148.960
C07089=1150.149,417.036,-89.350,-176.226,9.933,148.959
C07090=1150.146,416.816,-89.317,-176.225,9.932,148.959
C07091=1150.145,416.595,-89.284,-176.225,9.930,148.958
C07092=1150.143,416.373,-89.251,-176.224,9.928,148.958
C07093=1150.142,416.151,-89.219,-176.224,9.927,148.957
C07094=1150.142,415.931,-89.186,-176.223,9.925,148.957
C07095=1150.143,415.708,-89.154,-176.223,9.923,148.956
C07096=1150.144,415.487,-89.121,-176.222,9.922,148.955
C07097=1150.145,415.240,-89.084,-176.221,9.920,148.955
C07098=1150.148,414.993,-89.048,-176.221,9.918,148.954
C07099=1150.151,414.745,-89.011,-176.221,9.916,148.953
C07100=1150.155,414.498,-88.974,-176.220,9.914,148.953
C07101=1150.159,414.251,-88.937,-176.219,9.912,148.952
C07102=1150.162,414.004,-88.899,-176.218,9.910,148.951
C07103=1150.166,413.756,-88.862,-176.218,9.909,148.951
C07104=1150.170,413.509,-88.826,-176.217,9.907,148.950
C07105=1150.174,413.262,-88.789,-176.216,9.905,148.949
C07106=1150.178,413.015,-88.752,-176.216,9.902,148.949
C07107=1150.181,412.767,-88.715,-176.215,9.900,148.948
C07108=1150.185,412.520,-88.678,-176.215,9.899,148.947
C07109=1150.189,412.273,-88.642,-176.214,9.897,148.946
C07110=1150.194,412.026,-88.605,-176.213,9.895,148.946
C07111=1150.197,411.778,-88.567,-176.212,9.893,148.945
C07112=1150.201,411.531,-88.530,-176.211,9.891,148.945
C07113=1150.204,411.284,-88.494,-176.210,9.889,148.944
C07114=1150.208,411.037,-88.457,-176.210,9.888,148.943
C07115=1150.212,410.790,-88.420,-176.209,9.886,148.942
C07116=1150.216,410.542,-88.383,-176.208,9.884,148.942
C07117=1150.220,410.295,-88.346,-176.207,9.882,148.941
C07118=1150.224,410.048,-88.309,-176.207,9.880,148.940
C07119=1150.228,409.800,-88.272,-176.206,9.879,148.940
C07120=1150.231,409.554,-88.236,-176.205,9.876,148.939
C07121=1150.235,409.306,-88.199,-176.204,9.875,148.938
C07122=1150.239,409.059,-88.161,-176.203,9.873,148.938
C07123=1150.243,408.812,-88.124,-176.202,9.871,148.937
C07124=1150.247,408.565,-88.087,-176.202,9.869,148.936
C07125=1150.251,408.318,-88.050,-176.201,9.867,148.935
C07126=1150.254,408.070,-88.014,-176.200,9.865,148.935
C07127=1150.258,407.823,-87.977,-176.199,9.864,148.934
C07128=1150.262,407.576,-87.940,-176.198,9.862,148.933
C07129=1150.266,407.328,-87.903,-176.197,9.860,148.933
C07130=1150.270,407.081,-87.866,-176.196,9.858,148.932
C07131=1150.274,406.833,-87.829,-176.196,9.856,148.931
C07132=1150.277,406.586,-87.793,-176.195,9.854,148.930
C07133=1150.281,406.339,-87.756,-176.194,9.852,148.930
C07134=1150.285,406.093,-87.718,-176.193,9.850,148.929
C07135=1150.288,405.845,-87.681,-176.191,9.849,148.928
C07136=1150.293,405.598,-87.644,-176.190,9.847,148.927
C07137=1150.297,405.350,-87.608,-176.190,9.845,148.927
C07138=1150.300,405.104,-87.571,-176.189,9.843,148.926
C07139=1150.304,404.856,-87.534,-176.188,9.842,148.925
C07140=1150.308,404.608,-87.497,-176.187,9.839,148.924
C07141=1150.312,404.361,-87.460,-176.186,9.838,148.924
C07142=1150.316,404.114,-87.423,-176.185,9.836,148.923
C07143=1150.320,403.867,-87.387,-176.184,9.834,148.922
C07144=1150.323,403.620,-87.350,-176.183,9.832,148.921
C07145=1150.327,403.372,-87.313,-176.182,9.830,148.921
C07146=1150.330,403.126,-87.276,-176.181,9.828,148.920
C07147=1150.335,402.878,-87.239,-176.180,9.826,148.919
C07148=1150.339,402.631,-87.202,-176.179,9.824,148.918
C07149=1150.343,402.384,-87.165,-176.178,9.823,148.917
C07150=1150.346,402.136,-87.128,-176.177,9.821,148.917
C07151=1150.350,401.889,-87.091,-176.176,9.819,148.916
C07152=1150.354,401.642,-87.055,-176.175,9.817,148.915
C07153=1150.358,401.395,-87.018,-176.174,9.815,148.914
C07154=1150.362,401.148,-86.981,-176.173,9.813,148.914
C07155=1150.365,400.900,-86.944,-176.172,9.811,148.913
C07156=1150.369,400.653,-86.907,-176.171,9.809,148.912
C07157=1150.373,400.406,-86.871,-176.170,9.807,148.911
C07158=1150.377,400.158,-86.834,-176.169,9.805,148.910
C07159=1150.381,399.911,-86.797,-176.168,9.803,148.910
C07160=1150.384,399.664,-86.759,-176.167,9.801,148.909
C07161=1150.388,399.417,-86.723,-176.166,9.799,148.908
C07162=1150.392,399.170,-86.686,-176.165,9.797,148.907
C07163=1150.396,398.923,-86.649,-176.164,9.795,148.906
C07164=1150.400,398.676,-86.612,-176.163,9.793,148.906
C07165=1150.403,398.428,-86.575,-176.162,9.791,148.905
C07166=1150.407,398.180,-86.538,-176.160,9.789,148.904
C07167=1150.411,397.934,-86.502,-176.160,9.786,148.903
C07168=1150.415,397.686,-86.465,-176.159,9.784,148.902
C07169=1150.419,397.439,-86.428,-176.158,9.782,148.902
C07170=1150.422,397.191,-86.391,-176.157,9.780,148.901
C07171=1150.427,396.944,-86.354,-176.156,9.778,148.900
C07172=1150.431,396.697,-86.317,-176.155,9.776,148.899
C07173=1150.434,396.450,-86.281,-176.154,9.774,148.898
C07174=1150.438,396.203,-86.244,-176.153,9.771,148.897
C07175=1150.441,395.956,-86.206,-176.152,9.769,148.896
C07176=1150.445,395.708,-86.169,-176.151,9.767,148.896
C07177=1150.449,395.461,-86.132,-176.150,9.765,148.895
C07178=1150.454,395.214,-86.095,-176.150,9.762,148.894
C07179=1150.457,394.967,-86.059,-176.149,9.760,148.893
C07180=1150.460,394.719,-86.022,-176.147,9.758,148.892
C07181=1150.465,394.472,-85.985,-176.147,9.755,148.892
C07182=1150.469,394.225,-85.948,-176.146,9.753,148.891
C07183=1150.473,393.978,-85.911,-176.145,9.750,148.890
C07184=1150.476,393.731,-85.875,-176.144,9.748,148.889
C07185=1150.480,393.483,-85.838,-176.144,9.747,148.888
C07186=1150.484,393.236,-85.801,-176.143,9.744,148.887
C07187=1150.488,392.989,-85.764,-176.142,9.742,148.887
C07188=1150.492,392.741,-85.727,-176.141,9.739,148.886
C07189=1150.495,392.494,-85.691,-176.141,9.736,148.885
C07190=1150.499,392.247,-85.654,-176.140,9.734,148.884
C07191=1150.503,391.999,-85.617,-176.139,9.731,148.883
C07192=1150.507,391.752,-85.580,-176.139,9.728,148.882
C07193=1150.511,391.466,-85.537,-176.138,9.725,148.881
C07194=1150.515,391.179,-85.495,-176.138,9.722,148.880
C07195=1150.519,390.893,-85.452,-176.137,9.719,148.879
C07196=1150.524,390.606,-85.409,-176.136,9.716,148.878
C07197=1150.528,390.359,-85.372,-176.136,9.713,148.877
C07198=1150.532,390.112,-85.336,-176.135,9.711,148.877
C07199=1150.535,389.865,-85.299,-176.135,9.708,148.876
C07200=1150.540,389.618,-85.262,-176.134,9.705,148.875
C07201=1150.543,389.370,-85.225,-176.134,9.702,148.874
C07202=1150.547,389.123,-85.188,-176.134,9.700,148.873
C07203=1150.551,388.876,-85.151,-176.133,9.697,148.872
C07204=1150.555,388.629,-85.115,-176.133,9.694,148.872
C07205=1150.559,388.382,-85.078,-176.133,9.691,148.871
C07206=1150.563,388.134,-85.041,-176.132,9.689,148.870
C07207=1150.566,387.886,-85.004,-176.133,9.685,148.869
C07208=1150.570,387.640,-84.968,-176.132,9.682,148.868
C07209=1150.574,387.392,-84.931,-176.132,9.679,148.868
C07210=1150.578,387.145,-84.894,-176.132,9.676,148.867
C07211=1150.582,386.898,-84.857,-176.132,9.673,148.866
C07212=1150.585,386.651,-84.821,-176.132,9.670,148.865
C07213=1150.589,386.403,-84.784,-176.132,9.666,148.864
C07214=1150.593,386.156,-84.747,-176.132,9.664,148.864
C07215=1150.597,385.908,-84.711,-176.132,9.660,148.863
C07216=1150.601,385.661,-84.675,-176.133,9.657,148.862
C07217=1150.605,385.414,-84.638,-176.133,9.653,148.861
C07218=1150.609,385.167,-84.601,-176.134,9.650,148.860
C07219=1150.612,384.919,-84.564,-176.134,9.647,148.860
C07220=1150.616,384.672,-84.527,-176.135,9.643,148.859
C07221=1150.620,384.425,-84.491,-176.135,9.640,148.858
C07222=1150.624,384.178,-84.454,-176.136,9.636,148.857
C07223=1150.627,383.931,-84.417,-176.136,9.633,148.857
C07224=1150.632,383.683,-84.381,-176.137,9.630,148.856
C07225=1150.636,383.436,-84.344,-176.137,9.626,148.855
C07226=1150.639,383.189,-84.308,-176.138,9.622,148.854
C07227=1150.643,382.941,-84.271,-176.139,9.619,148.853
C07228=1150.647,382.694,-84.234,-176.140,9.615,148.853
C07229=1150.650,382.447,-84.198,-176.140,9.611,148.852
C07230=1150.654,382.199,-84.162,-176.142,9.607,148.851
C07231=1150.658,381.952,-84.125,-176.142,9.604,148.851
C07232=1150.662,381.705,-84.089,-176.143,9.600,148.850
C07233=1150.666,381.458,-84.052,-176.145,9.596,148.849
C07234=1150.670,381.211,-84.015,-176.146,9.592,148.848
C07235=1150.674,380.963,-83.979,-176.147,9.589,148.848
C07236=1150.677,380.715,-83.942,-176.148,9.585,148.847
C07237=1150.681,380.469,-83.906,-176.149,9.581,148.846
C07238=1150.685,380.221,-83.870,-176.151,9.577,148.846
C07239=1150.689,379.974,-83.833,-176.152,9.573,148.845
C07240=1150.692,379.727,-83.797,-176.154,9.569,148.845
C07241=1150.696,379.479,-83.760,-176.155,9.565,148.844
C07242=1150.700,379.232,-83.724,-176.157,9.561,148.843
C07243=1150.704,378.985,-83.687,-176.158,9.557,148.843
C07244=1150.708,378.738,-83.650,-176.160,9.554,148.842
C07245=1150.712,378.490,-83.615,-176.161,9.550,148.842
C07246=1150.716,378.243,-83.578,-176.163,9.545,148.841
C07247=1150.720,377.995,-83.543,-176.165,9.541,148.840
C07248=1150.724,377.748,-83.506,-176.166,9.537,148.840
C07249=1150.727,377.501,-83.469,-176.168,9.534,148.839
C07250=1150.732,377.254,-83.433,-176.170,9.529,148.839
C07251=1150.735,377.007,-83.397,-176.172,9.525,148.838
C07252=1150.739,376.759,-83.361,-176.174,9.521,148.837
C07253=1150.743,376.512,-83.325,-176.176,9.517,148.837
C07254=1150.747,376.264,-83.288,-176.177,9.513,148.836
C07255=1150.750,376.017,-83.252,-176.179,9.509,148.836
C07256=1150.755,375.769,-83.216,-176.181,9.504,148.835
C07257=1150.758,375.523,-83.180,-176.183,9.501,148.835
C07258=1150.763,375.275,-83.144,-176.185,9.497,148.834
C07259=1150.766,375.028,-83.107,-176.187,9.493,148.834
C07260=1150.770,374.780,-83.071,-176.189,9.488,148.833
C07261=1150.774,374.533,-83.035,-176.191,9.485,148.833
C07262=1150.777,374.286,-82.999,-176.193,9.480,148.832
C07263=1150.782,374.038,-82.963,-176.195,9.476,148.832
C07264=1150.785,373.791,-82.927,-176.198,9.472,148.831
C07265=1150.790,373.543,-82.891,-176.200,9.468,148.831
C07266=1150.793,373.296,-82.855,-176.202,9.464,148.830
C07267=1150.797,373.049,-82.819,-176.205,9.460,148.830
C07268=1150.801,372.801,-82.783,-176.207,9.456,148.829
C07269=1150.805,372.554,-82.747,-176.209,9.452,148.829
C07270=1150.809,372.306,-82.710,-176.212,9.447,148.828
C07271=1150.812,372.059,-82.675,-176.213,9.444,148.828
C07272=1150.816,371.811,-82.639,-176.216,9.439,148.828
C07273=1150.820,371.564,-82.603,-176.218,9.435,148.827
C07274=1150.824,371.317,-82.567,-176.220,9.431,148.827
C07275=1150.828,371.070,-82.532,-176.223,9.427,148.826
C07276=1150.832,370.822,-82.496,-176.225,9.422,148.826
C07277=1150.836,370.575,-82.460,-176.227,9.419,148.825
C07278=1150.840,370.328,-82.424,-176.230,9.414,148.825
C07279=1150.843,370.080,-82.388,-176.233,9.410,148.825
C07280=1150.848,369.832,-82.352,-176.235,9.406,148.824
C07281=1150.851,369.585,-82.317,-176.237,9.402,148.824
C07282=1150.855,369.338,-82.281,-176.239,9.398,148.823
C07283=1150.859,369.091,-82.246,-176.242,9.394,148.823
C07284=1150.864,368.843,-82.210,-176.244,9.390,148.822
C07285=1150.867,368.595,-82.174,-176.247,9.386,148.822
C07286=1150.871,368.348,-82.139,-176.250,9.382,148.822
C07287=1150.875,368.100,-82.103,-176.252,9.377,148.821
C07288=1150.878,367.853,-82.067,-176.254,9.374,148.821
C07289=1150.883,367.606,-82.031,-176.257,9.370,148.821
C07290=1150.887,367.359,-81.996,-176.259,9.365,148.820
C07291=1150.891,367.111,-81.961,-176.262,9.361,148.820
C07292=1150.894,366.863,-81.925,-176.264,9.358,148.819
C07293=1150.898,366.616,-81.890,-176.267,9.354,148.819
C07294=1150.902,366.369,-81.854,-176.270,9.349,148.819
C07295=1150.906,366.121,-81.819,-176.272,9.345,148.818
C07296=1150.910,365.873,-81.783,-176.274,9.342,148.818
C07297=1150.914,365.590,-81.743,-176.278,9.337,148.818
C07298=1150.919,365.308,-81.702,-176.280,9.332,148.817
C07299=1150.923,365.024,-81.661,-176.284,9.327,148.817
C07300=1150.928,364.741,-81.621,-176.286,9.323,148.816
C07301=1150.931,364.494,-81.585,-176.289,9.319,148.816
C07302=1150.936,364.247,-81.550,-176.292,9.314,148.816
C07303=1150.940,363.999,-81.515,-176.294,9.311,148.815
C07304=1150.943,363.751,-81.479,-176.296,9.307,148.815
C07305=1150.947,363.504,-81.444,-176.299,9.303,148.815
C07306=1150.951,363.257,-81.409,-176.302,9.298,148.814
C07307=1150.955,363.009,-81.374,-176.304,9.295,148.814
C07308=1150.959,362.761,-81.338,-176.307,9.291,148.814
C07309=1150.963,362.514,-81.303,-176.310,9.286,148.813
C07310=1150.967,362.266,-81.268,-176.312,9.283,148.813
C07311=1150.971,362.019,-81.233,-176.314,9.279,148.813
C07312=1150.974,361.771,-81.197,-176.317,9.275,148.812
C07313=1150.979,361.524,-81.163,-176.320,9.271,148.812
C07314=1150.983,361.276,-81.127,-176.322,9.267,148.812
C07315=1150.986,361.029,-81.092,-176.325,9.263,148.811
C07316=1150.991,360.781,-81.057,-176.327,9.260,148.811
C07317=1150.994,360.534,-81.022,-176.330,9.255,148.811
C07318=1150.998,360.286,-80.987,-176.333,9.251,148.810
C07319=1151.002,360.039,-80.952,-176.335,9.248,148.810
C07320=1151.006,359.792,-80.917,-176.338,9.244,148.810
C07321=1151.010,359.544,-80.882,-176.340,9.239,148.810
C07322=1151.014,359.297,-80.847,-176.342,9.236,148.809
C07323=1151.018,359.049,-80.812,-176.345,9.232,148.809
